VAR CONSTANT
	NULL:                                   			XWORD := 0;
	data:						iol_slave_bis00lh_data;			(*$	Parameters struct variable	$*)
	CONVERSION_this:			iol_slave;						(*$ Instance to which the method applies $*)
	
END_VAR



(*** Start parameter configuration ***)

(* STANDARD PARAMETERS CONFIGURATION *)

(* RMH RFID TEST *)
rfid_input_bitheader_1.CP := rfid_input_buffer.ByteArr[0].0;
rfid_input_bitheader_1.AA := rfid_input_buffer.ByteArr[0].1;
rfid_input_bitheader_1.AE := rfid_input_buffer.ByteArr[0].2;
rfid_input_bitheader_1.AF := rfid_input_buffer.ByteArr[0].3;
rfid_input_bitheader_1.Bit4 := rfid_input_buffer.ByteArr[0].4;
rfid_input_bitheader_1._TO := rfid_input_buffer.ByteArr[0].5;
rfid_input_bitheader_1.HF := rfid_input_buffer.ByteArr[0].6;
rfid_input_bitheader_1.BB := rfid_input_buffer.ByteArr[0].7;

rfid_input_bitheader_2.CP := rfid_input_buffer.ByteArr[0].0;
rfid_input_bitheader_2.AA := rfid_input_buffer.ByteArr[0].1;
rfid_input_bitheader_2.AE := rfid_input_buffer.ByteArr[0].2;
rfid_input_bitheader_2.AF := rfid_input_buffer.ByteArr[0].3;
rfid_input_bitheader_2.Bit4 := rfid_input_buffer.ByteArr[0].4;
rfid_input_bitheader_2._TO := rfid_input_buffer.ByteArr[0].5;
rfid_input_bitheader_2.HF := rfid_input_buffer.ByteArr[0].6;
rfid_input_bitheader_2.BB := rfid_input_buffer.ByteArr[0].7;

rfid_output_bitheader_1.TI := rfid_output_buffer.ByteArr[0].0;
rfid_output_bitheader_1.Bit1 := rfid_output_buffer.ByteArr[0].1;
rfid_output_bitheader_1.GR := rfid_output_buffer.ByteArr[0].2;
rfid_output_bitheader_1.Bit3 := rfid_output_buffer.ByteArr[0].3;
rfid_output_bitheader_1.Bit4 := rfid_output_buffer.ByteArr[0].4;
rfid_output_bitheader_1.KA := rfid_output_buffer.ByteArr[0].5;
rfid_output_bitheader_1.TI := rfid_output_buffer.ByteArr[0].6;
rfid_output_bitheader_1.Bit7 := rfid_output_buffer.ByteArr[0].7;

rfid_output_bitheader_2.TI := rfid_output_buffer.ByteArr[0].0;
rfid_output_bitheader_2.Bit1 := rfid_output_buffer.ByteArr[0].1;
rfid_output_bitheader_2.GR := rfid_output_buffer.ByteArr[0].2;
rfid_output_bitheader_2.Bit3 := rfid_output_buffer.ByteArr[0].3;
rfid_output_bitheader_2.Bit4 := rfid_output_buffer.ByteArr[0].4;
rfid_output_bitheader_2.KA := rfid_output_buffer.ByteArr[0].5;
rfid_output_bitheader_2.TI := rfid_output_buffer.ByteArr[0].6;
rfid_output_bitheader_2.Bit7 := rfid_output_buffer.ByteArr[0].7;


(*IF iol_slave_is_not_initialized(CONVERSION_this := CONVERSION_this)
	OR
	iol_slave_is_configured(CONVERSION_this := CONVERSION_this)
THEN
	RETURN;
END_IF


iol_slave_configure_parameter(
	current_value_address := ADR(CONVERSION_this.vendor_name),
	configured_value_address := NULL,
	length := SIZEOF(CONVERSION_this.vendor_name),
	_type := ADST_STRING,
	coe_index := 16#0010,
	coe_sub_index := 16#00,
	readable := TRUE,
	writeable := FALSE,
	to_check := FALSE,
	CONVERSION_this := CONVERSION_this);


iol_slave_configure_parameter(
	current_value_address := ADR(CONVERSION_this.product_name),
	configured_value_address := NULL,
	length := SIZEOF(CONVERSION_this.product_name),
	_type := ADST_STRING,
	coe_index := 16#0012,
	coe_sub_index := 16#00,
	readable := TRUE,
	writeable := FALSE,
	to_check := FALSE,
	CONVERSION_this := CONVERSION_this);

iol_slave_configure_parameter(
	current_value_address := ADR(CONVERSION_this.product_id),
	configured_value_address := NULL,
	length := SIZEOF(CONVERSION_this.product_id),
	_type := ADST_STRING,
	coe_index := 16#0013,
	coe_sub_index := 16#00,
	readable := TRUE,
	writeable := FALSE,
	to_check := FALSE,
	CONVERSION_this := CONVERSION_this);


iol_slave_configure_parameter(
	current_value_address := ADR(CONVERSION_this.hardware_revision),
	configured_value_address := NULL,
	length := SIZEOF(CONVERSION_this.hardware_revision),
	_type := ADST_STRING,
	coe_index := 16#0016,
	coe_sub_index := 16#00,
	readable := TRUE,
	writeable := FALSE,
	to_check := FALSE,
	CONVERSION_this := CONVERSION_this);

iol_slave_configure_parameter(
	current_value_address := ADR(CONVERSION_this.firmware_revision),
	configured_value_address := NULL,
	length := SIZEOF(CONVERSION_this.firmware_revision),
	_type := ADST_STRING,
	coe_index := 16#0017,
	coe_sub_index := 16#00,
	readable := TRUE,
	writeable := FALSE,
	to_check := FALSE,
	CONVERSION_this := CONVERSION_this);

iol_slave_configure_parameter(
	current_value_address := ADR(CONVERSION_this.current_app_specific_tag),
	configured_value_address := ADR(CONVERSION_this.configured_app_specific_tag),
	length := SIZEOF(CONVERSION_this.current_app_specific_tag),
	_type := ADST_STRING,
	coe_index := 16#0018,
	coe_sub_index := 16#00,
	readable := TRUE,
	writeable := TRUE,
	to_check := TRUE,
	CONVERSION_this := CONVERSION_this);
	
	

(* CUSTOM PARAMETERS CONFIGURATION *)
(*
iol_slave_configure_parameter(
	current_value_address := ADR(data.v_param_1),
	configured_value_address := ADR(data.v_param_1),
	length := SIZEOF(data.v_param_1),
	_type := ADST_UINT8,
	coe_index := 16#0040,
	coe_sub_index := 16#01,
	readable := TRUE,
	writeable := TRUE,
	to_check := FALSE,
	CONVERSION_this := CONVERSION_this);
	
iol_slave_configure_parameter(
	current_value_address := ADR(data.v_param_2),
	configured_value_address := ADR(data.v_param_2),
	length := SIZEOF(data.v_param_2),
	_type := ADST_UINT8,
	coe_index := 16#0040,
	coe_sub_index := 16#02,
	readable := TRUE,
	writeable := TRUE,
	to_check := FALSE,
	CONVERSION_this := CONVERSION_this);
	
iol_slave_configure_parameter(
	current_value_address := ADR(data.v_param_3),
	configured_value_address := ADR(data.v_param_3),
	length := SIZEOF(data.v_param_3),
	_type := ADST_UINT8,
	coe_index := 16#0040,
	coe_sub_index := 16#03,
	readable := TRUE,
	writeable := TRUE,
	to_check := FALSE,
	CONVERSION_this := CONVERSION_this);
	
iol_slave_configure_parameter(
	current_value_address := ADR(data.v_param_4),
	configured_value_address := ADR(data.v_param_4),
	length := SIZEOF(data.v_param_4),
	_type := ADST_UINT8,
	coe_index := 16#0040,
	coe_sub_index := 16#04,
	readable := TRUE,
	writeable := TRUE,
	to_check := FALSE,
	CONVERSION_this := CONVERSION_this);
	
iol_slave_configure_parameter(
	current_value_address := ADR(data.v_param_5),
	configured_value_address := ADR(data.v_param_5),
	length := SIZEOF(data.v_param_5),
	_type := ADST_UINT8,
	coe_index := 16#0040,
	coe_sub_index := 16#05,
	readable := TRUE,
	writeable := TRUE,
	to_check := FALSE,
	CONVERSION_this := CONVERSION_this);
	
iol_slave_configure_parameter(
	current_value_address := ADR(data.v_param_6),
	configured_value_address := ADR(data.v_param_6),
	length := SIZEOF(data.v_param_6),
	_type := ADST_UINT8,
	coe_index := 16#0040,
	coe_sub_index := 16#06,
	readable := TRUE,
	writeable := TRUE,
	to_check := FALSE,
	CONVERSION_this := CONVERSION_this);
	*)
	

	
CONVERSION_this.CONVERSION_private.last_info_data_index := 6;

(*** End parameter configuration ***)
iol_slave_configuration_completed(
	parameters_ptr := ADR(data),
	parameters_struct_size := SIZEOF(data),
	CONVERSION_this := CONVERSION_this);*)

END_FUNCTION

// ---- POUs/AFL extensions/IO_Link/FUN/iol_slave_ray26p_configure.TcPOU
(*$
<p>This function configures a generic <a target="_blank" href="#iol_slave">iol_slave</a> as a <strong>Sick WTB2SC - 2P3244</strong>. It allow to connect the object to the device-specific
parameters structure variable <a target="_blank" href="#iol_slave_wtb2sc_data">iol_slave_wtb2sc_data</a>.</p>
<p>This function should be called at startup only.</p>
$*)

FUNCTION iol_slave_ray26p_configure : VOID
VAR_IN_OUT
	data:					iol_slave_ray26p_data;			(*$	Parameters struct variable$*)
	CONVERSION_this:		iol_slave;						(*$ Instance to which the method applies $*)
END_VAR

VAR CONSTANT
	NULL:                                   			XWORD := 0;
END_VAR

IF iol_slave_is_not_initialized(CONVERSION_this := CONVERSION_this)
	OR
	iol_slave_is_configured(CONVERSION_this := CONVERSION_this)
THEN
	RETURN;
END_IF

(*** Start parameter configuration ***)

(* STANDARD PARAMETERS CONFIGURATION *)

iol_slave_configure_parameter(
	current_value_address := ADR(CONVERSION_this.vendor_name),
	configured_value_address := NULL,
	length := SIZEOF(CONVERSION_this.vendor_name),
	_type := ADST_STRING,
	coe_index := 16#0010,
	coe_sub_index := 16#00,
	readable := TRUE,
	writeable := FALSE,
	to_check := FALSE,
	CONVERSION_this := CONVERSION_this);

iol_slave_configure_parameter(
	current_value_address := ADR(CONVERSION_this.product_name),
	configured_value_address := NULL,
	length := SIZEOF(CONVERSION_this.product_name),
	_type := ADST_STRING,
	coe_index := 16#0012,
	coe_sub_index := 16#00,
	readable := TRUE,
	writeable := FALSE,
	to_check := FALSE,
	CONVERSION_this := CONVERSION_this);

iol_slave_configure_parameter(
	current_value_address := ADR(CONVERSION_this.product_id),
	configured_value_address := NULL,
	length := SIZEOF(CONVERSION_this.product_id),
	_type := ADST_STRING,
	coe_index := 16#0013,
	coe_sub_index := 16#00,
	readable := TRUE,
	writeable := FALSE,
	to_check := FALSE,
	CONVERSION_this := CONVERSION_this);


iol_slave_configure_parameter(
	current_value_address := ADR(CONVERSION_this.hardware_revision),
	configured_value_address := NULL,
	length := SIZEOF(CONVERSION_this.hardware_revision),
	_type := ADST_STRING,
	coe_index := 16#0016,
	coe_sub_index := 16#00,
	readable := TRUE,
	writeable := FALSE,
	to_check := FALSE,
	CONVERSION_this := CONVERSION_this);

iol_slave_configure_parameter(
	current_value_address := ADR(CONVERSION_this.firmware_revision),
	configured_value_address := NULL,
	length := SIZEOF(CONVERSION_this.firmware_revision),
	_type := ADST_STRING,
	coe_index := 16#0017,
	coe_sub_index := 16#00,
	readable := TRUE,
	writeable := FALSE,
	to_check := FALSE,
	CONVERSION_this := CONVERSION_this);


(* CUSTOM PARAMETERS CONFIGURATION *)

iol_slave_configure_parameter(
	current_value_address := ADR(data.teach_in_state),
	configured_value_address := NULL,
	length := SIZEOF(data.teach_in_state),
	_type := ADST_UINT8,
	coe_index := 16#003B,
	coe_sub_index :=16#00,
	readable := TRUE,
	writeable := FALSE,
	to_check := FALSE,
	CONVERSION_this := CONVERSION_this);
	
iol_slave_configure_parameter(
	current_value_address := ADR(data.teach_in_channel),
	configured_value_address := ADR(data.teach_in_channel),
	length := SIZEOF(data.teach_in_channel),
	_type := ADST_UINT8,
	coe_index := 16#003A,
	coe_sub_index :=16#00,
	readable := TRUE,
	writeable := TRUE,
	to_check := TRUE, (* to be evaluated *)
	CONVERSION_this := CONVERSION_this);
	
iol_slave_configure_parameter(
	current_value_address := ADR(data.sender_configuration),
	configured_value_address := ADR(data.sender_configuration),
	length := SIZEOF(data.sender_configuration),
	_type := ADST_UINT8,
	coe_index := 16#0061,
	coe_sub_index :=16#00,
	readable := TRUE,
	writeable := TRUE,
	to_check := TRUE, (* to be evaluated *)
	CONVERSION_this := CONVERSION_this);
	
iol_slave_configure_parameter(
	current_value_address := ADR(data.Pin2_configuration),
	configured_value_address := ADR(data.Pin2_configuration),
	length := SIZEOF(data.Pin2_configuration),
	_type := ADST_UINT8,
	coe_index := 16#0079,
	coe_sub_index :=16#00,
	readable := TRUE,
	writeable := TRUE,
	to_check := TRUE, (* to be evaluated *)
	CONVERSION_this := CONVERSION_this);

iol_slave_configure_parameter(
	current_value_address := ADR(data.quality_of_teach),
	configured_value_address := NULL,
	length := SIZEOF(data.quality_of_teach),
	_type := ADST_UINT8,
	coe_index := 16#0072,
	coe_sub_index :=16#00,
	readable := TRUE,
	writeable := FALSE,
	to_check := FALSE, (* to be evaluated *)
	CONVERSION_this := CONVERSION_this);
	
iol_slave_configure_parameter(
	current_value_address := ADR(data.system_state),
	configured_value_address := NULL,
	length := SIZEOF(data.system_state),
	_type := ADST_UINT8,
	coe_index := 16#00E2,
	coe_sub_index :=16#00,
	readable := TRUE,
	writeable := FALSE,
	to_check := FALSE, (* to be evaluated *)
	CONVERSION_this := CONVERSION_this);


CONVERSION_this.CONVERSION_private.last_info_data_index := 5;

(*** End parameter configuration ***)

iol_slave_configuration_completed(
	parameters_ptr := ADR(data),
	parameters_struct_size := SIZEOF(data),
	CONVERSION_this := CONVERSION_this);

END_FUNCTION

// ---- Application/CSP/Customer Interface/csp_customerInterfaces_old.TcPOU
 (*********************************** G.D S.p.A. - Technical Department ***********************************
============= PROGRAM INFO ============
FOLDER:             TBD
MACHINES INVOLVED:  TBD 

============= DESCRIPTION =============
Exit unit device declaration

============= REVISIONS ===============
Date		Version	 	Author      	Description             
----------	-------		------------  	--------------------------------------------
2019/03/27 	0000.00	 	CEC 			Creation of the PRG

**********************************************************************************************************)
(*$R process_ref:= prc; $*)

PROGRAM csp_customerInterfaces_old

VAR
	prc:								process;
	prc_path:							STRING;
	
	CasePacker:							csp_customerInterfaces_casePacker;
	Palletizer:							csp_customerInterfaces_palletizer;
	
END_VAR

VAR PERSISTENT
	Order:								csp_customerInterfaces_order;
	Product:							csp_customerInterfaces_product;
	Recipe:								csp_customerInterfaces_recipe;														
	Material:							ARRAY [0..14] OF csp_customerInterfaces_material;
	Mark:								csp_customerInterfaces_mark;
	NextOrder:							csp_customerInterfaces_order;	
	NextProduct:						csp_customerInterfaces_product;	
	NextRecipe:							csp_customerInterfaces_recipe;		
	NextMaterial:						ARRAY [0..14] OF csp_customerInterfaces_material;			
	MES:								csp_customerInterfaces_MES;	
		
END_VAR

_read_var_input();

_objects_manager();

IF NOT objects_running()
THEN
	RETURN;	
END_IF

_read_process_image();

_mode_manager();

CASE process_get_mode(prc) of
	MODE_ABSENT,
	MODE_INACTIVE:
		RETURN;
	MODE_TEST:
		_handle_process_test();
END_CASE

_set_runtime_properties();

(********************************* BODY *********************************)


(* CSP STATUS *)

Dock();
//CasePacker.Status.Online := machine_is_operational(csp.mch); 
//CasePacker.Status.Job := csp_main_brand.p_carton_format;
//CasePacker.Status.NextJob := // need to figure out next job
CasePacker.Status.Running := machine_is_running(csp.mch);

CasePacker.Status.Faulted.Main := machine_is_stopped(csp.mch)
									AND csp_main_interface.alarm_id_from_python <> 363 // CYCLE STOP FOR CASE SIDE
									AND csp_main_interface.alarm_id_from_python <> 622 // CYCLE STOP FOR TRANSFER SIDE
									AND csp_main_interface.alarm_id <> 363 // CYCLE STOP FOR CASE SIDE
									AND csp_main_interface.alarm_id <> 622; // CYCLE STOP FOR TRANSFER SIDE
									
CasePacker.Status.Faulted.CaseBlanks := csp_case_feed_magazine.AML_Faulted;

//CasePacker.Status.RunOut := csp_main_motorization.empty_command;
//CasePacker.Status.RunOutComplete := message_is_on(csp_case_virtualMaster.runout_complete);

CasePacker.Status.Rate.Target := LREAL_TO_INT(csp_main_motorization_manager.motm.actual_velocity_setpoint);
CasePacker.Status.Rate.Actual := LREAL_TO_INT(csp_main_motorization_manager.motm.actual_velocity);

CasePacker.Status.Stop.AutoReason := csp_main_interface.alarm_id; 
CasePacker.Status.Stop.Estop := machine_is_stop_emergency_active(csp.mch);
CasePacker.Status.Stop.Guard := NOT safety_integrated_series_is_safely_closed(csp_case_main_safety_guards.sis) OR NOT safety_integrated_series_is_safely_closed(csp_transfer_main_safety_guards.sis);
CasePacker.Status.Stop.Operator := message_is_on(csp_case_main_services_pushbuttons.stop_dchk.alarm_asm.message);

CasePacker.Status.Starved.CaseBlanks := message_is_on(csp_case_feed_magazine_level_zonemin.magazine_level_zone_min_wem);
CasePacker.Status.Starved.Glue := NOT digital_input_is_active(csp_case_glue_hotmelt.level_ok_di);
//CasePacker.Status.Starved.Labels :=
CasePacker.Status.Starved.Units := csp_transfer_infeed_clamp.min_prime;

CasePacker.Status.Blocked.Downstream := message_is_on(csp_case_discharge_reject_sensors.downstream_backup_hold_aem);
CasePacker.Status.Blocked.Reject := message_is_on(csp_case_discharge_reject_sensors.consecutive_blocked_reject_aem);
CasePacker.Status.Blocked.Waste := message_is_on(csp_transfer_crosspusher_reject.backup_di_dchk.alarm_asm.message);




 
(*
CasePacker.Start.PeakWait :=
CasePacker.Start.Ramp:=
CasePacker.Start.Request:=
CasePacker.Production.GoodCasesNoReset:=
CasePacker.Production.GoodPods:=
CasePacker.Production.GoodPodsNoReset:=*)
CasePacker.Production.GoodUnits:= csp_case_main_statistics.logsect.hmi_shift_independent_sampled_counters.total_good_products; //log_section_get_total_good_production(csp_case_main_statistics.logsect);
(*CasePacker.Production.GoodUnitsNoReset:=
CasePacker.Production.PercentScrapUnits:=
CasePacker.Production.Rejects.Infeed_waterfall:=
CasePacker.Production.Rejects.Accumulator:=
CasePacker.Production.Rejects.Case_Feed:=*)
CasePacker.Production.Rejects.Discharge:= csp_case_discharge_reject.Discharge_reject_count;
(*CasePacker.Production.Rejects.TBD5:=
CasePacker.Production.Rejects.TBD6:= *)
CasePacker.Production.TotalScrapUnits:= csp_case_main_statistics.logsect.hmi_shift_independent_sampled_counters.total_rejected; //log_section_get_total_rejected(csp_case_main_statistics.logsect);
CasePacker.Production.TotalUnits:= (CasePacker.Production.GoodUnits + CasePacker.Production.TotalScrapUnits);
(*CasePacker.Production.TotalUnitsNoReset:=

CasePacker.CaseBlanks.ConsumedCart:=
CasePacker.CaseBlanks.ConsumedTotal:=
CasePacker.Labels.Consumed:=
CasePacker.CtCall.FaultedCaseSupply:=csp_case_feed_magazine.AML_Faulted;
CasePacker.CtCall.FaultedMain:=machine_is_stopped(csp.mch);
CasePacker.CtCall.FullScrapBin:=
CasePacker.CtCall.LowCaseSupply:=csp_case_feed_magazine.Magazine_low_level;
CasePacker.CtCall.LowGlueSupply:=csp_case_glue_hotmelt.level_ok_di;
//CasePacker.CtCall.LowLabelSupply:=.
CasePacker.CtCall.TBD1:=
CasePacker.CtCall.TBD2:=
CasePacker.CtCall.TBD3:=
CasePacker.Dock[1].Active:=
CasePacker.Dock[1].AmrExited:=
CasePacker.Dock[1].DropAvailable:=
CasePacker.Dock[1].EntryAck:=
CasePacker.Dock[1].EntryOK:=
CasePacker.Dock[1].EntryReq:=
CasePacker.Dock[1].PickAvailable:=
*)

(************************************************************************)

_handle_messages();

_write_output();

ACTION _handle_messages:
;
END_ACTION

ACTION _handle_process_test:
;
END_ACTION

ACTION _mode_manager:
IF process_mode_req_is_pending(prc)
THEN
    process_apply_mode_req_first_step(prc);
    CASE process_get_mode(prc) OF
        MODE_TO_ABSENT:
			;
        MODE_TO_INACTIVE:
			;
        MODE_TO_TEST:
			;
        MODE_TO_OPERATIONAL:
			;
    END_CASE
    process_apply_mode_req_second_step(prc);
END_IF
END_ACTION

ACTION _objects_manager:
IF objects_initialization()
THEN
	process_init(
		object_name					:= 'csp_customerInterfaces.prc', 
		machine						:= csp.mch, 
		CONVERSION_this				:= prc);
		
	prc_path 						:= process_get_path(prc);
END_IF

IF objects_running()
THEN
	process_cycle(prc);
END_IF
END_ACTION

ACTION _read_process_image:
;
END_ACTION

ACTION _read_var_input:
;
END_ACTION

ACTION _set_runtime_properties:
//CasePacker.Status.Online := TRUE;
END_ACTION

ACTION _write_output:
;
END_ACTION

ACTION Dock:
//Flexlink to AMR Dock 1
CasePacker.Dock[1].DropAvailable:= csp_case_feed_magazine.Flexlink_to_AMR_DropAvailable_1;
CasePacker.Dock[1].PickAvailable:= csp_case_feed_magazine.Flexlink_to_AMR_PickAvailable_1; 
CasePacker.Dock[1].Active:= csp_case_feed_magazine.Flexlink_to_AMR_Active_1;
CasePacker.Dock[1].EntryAck:= csp_case_feed_magazine.Flexlink_to_AMR_EntryAck_1;
CasePacker.Dock[1].EntryOK:= csp_case_feed_magazine.Flexlink_to_AMR_EntryOK_1;

(*csp_case_feed_magazine.AMR_to_Flexlink_EntryReq_1*) RAJ_to_Flexlink[3].0:= CasePacker.Dock[1].EntryReq;
(*csp_case_feed_magazine.AMR_to_Flexlink_AmrExited_1*) RAJ_to_Flexlink[3].1:= CasePacker.Dock[1].AmrExited;

//Flexlink to AMR Dock 2
CasePacker.Dock[2].DropAvailable:= csp_case_feed_magazine.Flexlink_to_AMR_DropAvailable_2;
CasePacker.Dock[2].PickAvailable:= csp_case_feed_magazine.Flexlink_to_AMR_PickAvailable_2; 
CasePacker.Dock[2].Active:= csp_case_feed_magazine.Flexlink_to_AMR_Active_2;
CasePacker.Dock[2].EntryAck:= csp_case_feed_magazine.Flexlink_to_AMR_EntryAck_2;
CasePacker.Dock[2].EntryOK:= csp_case_feed_magazine.Flexlink_to_AMR_EntryOK_2;

(*csp_case_feed_magazine.AMR_to_Flexlink_EntryReq_2*) RAJ_to_Flexlink[3].2:= CasePacker.Dock[2].EntryReq;
(*csp_case_feed_magazine.AMR_to_Flexlink_AmrExited_2*) RAJ_to_Flexlink[3].3:= CasePacker.Dock[2].AmrExited;

//Flexlink to AMR Dock 3
CasePacker.Dock[3].DropAvailable:= csp_case_feed_magazine.Flexlink_to_AMR_DropAvailable_3;
CasePacker.Dock[3].PickAvailable:= csp_case_feed_magazine.Flexlink_to_AMR_PickAvailable_3; 
CasePacker.Dock[3].Active:= csp_case_feed_magazine.Flexlink_to_AMR_Active_3;
CasePacker.Dock[3].EntryAck:= csp_case_feed_magazine.Flexlink_to_AMR_EntryAck_3;
CasePacker.Dock[3].EntryOK:= csp_case_feed_magazine.Flexlink_to_AMR_EntryOK_3;

(*csp_case_feed_magazine.AMR_to_Flexlink_EntryReq_3*) RAJ_to_Flexlink[3].4:= CasePacker.Dock[3].EntryReq;
(*csp_case_feed_magazine.AMR_to_Flexlink_AmrExited_3*) RAJ_to_Flexlink[3].5:= CasePacker.Dock[3].AmrExited;
END_ACTION

END_PROGRAM

// ---- Application/CSP/Customer Interface/csp_customerInterfaces_old_2.TcPOU
 (*********************************** G.D S.p.A. - Technical Department ***********************************
============= PROGRAM INFO ============
FOLDER:             TBD
MACHINES INVOLVED:  TBD 

============= DESCRIPTION =============
Exit unit device declaration

============= REVISIONS ===============
Date		Version	 	Author      	Description             
----------	-------		------------  	--------------------------------------------
2019/03/27 	0000.00	 	CEC 			Creation of the PRG

**********************************************************************************************************)
(*$R process_ref:= prc; $*)

PROGRAM csp_customerInterfaces_old_2

VAR
	prc:								process;
	prc_path:							STRING;
	
	Order:								csp_customerInterfaces_order;
	Product:							csp_customerInterfaces_product;
	Recipe:								csp_customerInterfaces_recipe;														
	Material:							ARRAY [0..14] OF csp_customerInterfaces_material;
	Mark:								csp_customerInterfaces_mark;
	NextOrder:							csp_customerInterfaces_order;	
	NextProduct:						csp_customerInterfaces_product;	
	NextRecipe:							csp_customerInterfaces_recipe;		
	NextMaterial:						ARRAY [0..14] OF csp_customerInterfaces_material;			
	MES:								csp_customerInterfaces_MES;		
	CasePacker:							csp_customerInterfaces_casePacker;
	Palletizer:							csp_customerInterfaces_palletizer;
	

END_VAR

_read_var_input();

_objects_manager();

IF NOT objects_running()
THEN
	RETURN;	
END_IF

_read_process_image();

_mode_manager();

CASE process_get_mode(prc) of
	MODE_ABSENT,
	MODE_INACTIVE:
		RETURN;
	MODE_TEST:
		_handle_process_test();
END_CASE

_set_runtime_properties();

(********************************* BODY *********************************)


(* CSP STATUS *)

CasePacker.Status.Online := machine_is_operational(csp.mch); 
CasePacker.Status.Job := csp_main_brand.p_carton_format;
//CasePacker.Status.NextJob := // need to figure out next job
CasePacker.Status.Running := machine_is_running(csp.mch);

CasePacker.Status.Faulted.Main := machine_is_stopped(csp.mch)
									AND csp_main_interface.alarm_id_from_python <> 363 // CYCLE STOP FOR CASE SIDE
									AND csp_main_interface.alarm_id_from_python <> 622; // CYCLE STOP FOR TRANSFER SIDE
CasePacker.Status.Faulted.CaseBlanks := csp_case_feed_magazine.AML_Faulted;

CasePacker.Status.RunOut := csp_main_motorization.empty_command;
CasePacker.Status.RunOutComplete := message_is_on(csp_case_virtualMaster.runout_complete);

CasePacker.Status.Rate.Target := LREAL_TO_INT(csp_main_motorization_manager.motm.actual_velocity_setpoint);
CasePacker.Status.Rate.Actual := LREAL_TO_INT(csp_main_motorization_manager.motm.actual_velocity);

CasePacker.Status.Stop.AutoReason := csp_main_interface.alarm_id; 
CasePacker.Status.Stop.Estop := machine_is_stop_emergency_active(csp.mch);
CasePacker.Status.Stop.Guard := NOT safety_integrated_series_is_safely_closed(csp_case_main_safety_guards.sis) OR NOT safety_integrated_series_is_safely_closed(csp_transfer_main_safety_guards.sis);
CasePacker.Status.Stop.Operator := message_is_on(csp_case_main_services_pushbuttons.stop_dchk.alarm_asm.message);

CasePacker.Status.Starved.CaseBlanks := message_is_on(csp_case_feed_magazine_level_zonemin.magazine_level_zone_min_aem);
CasePacker.Status.Starved.Glue := NOT digital_input_is_active(csp_case_glue_hotmelt.level_ok_di);
//CasePacker.Status.Starved.Labels :=
CasePacker.Status.Starved.Units := csp_transfer_infeed_clamp.min_prime;

CasePacker.Status.Blocked.Downstream := message_is_on(csp_case_discharge_reject_sensors.downstream_backup_hold_aem);
CasePacker.Status.Blocked.Reject := message_is_on(csp_case_discharge_reject_sensors.consecutive_blocked_reject_aem);
CasePacker.Status.Blocked.Waste := message_is_on(csp_transfer_crosspusher_reject.backup_di_dchk.alarm_asm.message);

//Flexlink to AMR Dock 1
CasePacker.Dock[1].DropAvailable:= csp_case_feed_magazine.Flexlink_to_AMR_DropAvailable_1;
CasePacker.Dock[1].PickAvailable:= csp_case_feed_magazine.Flexlink_to_AMR_PickAvailable_1; 
CasePacker.Dock[1].Active:= csp_case_feed_magazine.Flexlink_to_AMR_Active_1;
CasePacker.Dock[1].EntryAck:= csp_case_feed_magazine.Flexlink_to_AMR_EntryAck_1;
CasePacker.Dock[1].EntryOK:= csp_case_feed_magazine.Flexlink_to_AMR_EntryOK_1;

(*csp_case_feed_magazine.AMR_to_Flexlink_EntryReq_1*) RAJ_to_Flexlink[3].0:= CasePacker.Dock[1].EntryReq;
(*csp_case_feed_magazine.AMR_to_Flexlink_AmrExited_1*) RAJ_to_Flexlink[3].1:= CasePacker.Dock[1].AmrExited;

//Flexlink to AMR Dock 2
CasePacker.Dock[2].DropAvailable:= csp_case_feed_magazine.Flexlink_to_AMR_DropAvailable_2;
CasePacker.Dock[2].PickAvailable:= csp_case_feed_magazine.Flexlink_to_AMR_PickAvailable_2; 
CasePacker.Dock[2].Active:= csp_case_feed_magazine.Flexlink_to_AMR_Active_2;
CasePacker.Dock[2].EntryAck:= csp_case_feed_magazine.Flexlink_to_AMR_EntryAck_2;
CasePacker.Dock[2].EntryOK:= csp_case_feed_magazine.Flexlink_to_AMR_EntryOK_2;

(*csp_case_feed_magazine.AMR_to_Flexlink_EntryReq_2*) RAJ_to_Flexlink[3].2:= CasePacker.Dock[2].EntryReq;
(*csp_case_feed_magazine.AMR_to_Flexlink_AmrExited_2*) RAJ_to_Flexlink[3].3:= CasePacker.Dock[2].AmrExited;

//Flexlink to AMR Dock 3
CasePacker.Dock[3].DropAvailable:= csp_case_feed_magazine.Flexlink_to_AMR_DropAvailable_3;
CasePacker.Dock[3].PickAvailable:= csp_case_feed_magazine.Flexlink_to_AMR_PickAvailable_3; 
CasePacker.Dock[3].Active:= csp_case_feed_magazine.Flexlink_to_AMR_Active_3;
CasePacker.Dock[3].EntryAck:= csp_case_feed_magazine.Flexlink_to_AMR_EntryAck_3;
CasePacker.Dock[3].EntryOK:= csp_case_feed_magazine.Flexlink_to_AMR_EntryOK_3;

(*csp_case_feed_magazine.AMR_to_Flexlink_EntryReq_3*) RAJ_to_Flexlink[3].4:= CasePacker.Dock[3].EntryReq;
(*csp_case_feed_magazine.AMR_to_Flexlink_AmrExited_3*) RAJ_to_Flexlink[3].5:= CasePacker.Dock[3].AmrExited;




 
(*

CasePacker.Start.PeakWait :=
CasePacker.Start.Ramp:=
CasePacker.Start.Request:=

CasePacker.Production.GoodCasesNoReset:=
CasePacker.Production.GoodPods:=
CasePacker.Production.GoodPodsNoReset:=
CasePacker.Production.GoodUnits:=
CasePacker.Production.GoodUnitsNoReset:=
CasePacker.Production.PercentScrapUnits:=
CasePacker.Production.Rejects.TBD1:=
CasePacker.Production.Rejects.TBD2:=
CasePacker.Production.Rejects.TBD3:=
CasePacker.Production.Rejects.TBD4:=
CasePacker.Production.Rejects.TBD5:=
CasePacker.Production.Rejects.TBD6:=
CasePacker.Production.TotalScrapUnits:=
CasePacker.Production.TotalUnits:=
CasePacker.Production.TotalUnitsNoReset:=

CasePacker.CaseBlanks.ConsumedCart:=
CasePacker.CaseBlanks.ConsumedTotal:=

CasePacker.Labels.Consumed:=

CasePacker.CtCall.FaultedCaseSupply:=csp_case_feed_magazine.AML_Faulted;
CasePacker.CtCall.FaultedMain:=machine_is_stopped(csp.mch);
CasePacker.CtCall.FullScrapBin:=
CasePacker.CtCall.LowCaseSupply:=csp_case_feed_magazine.Magazine_low_level;
CasePacker.CtCall.LowGlueSupply:=csp_case_glue_hotmelt.level_ok_di;
//CasePacker.CtCall.LowLabelSupply:=.
CasePacker.CtCall.TBD1:=
CasePacker.CtCall.TBD2:=
CasePacker.CtCall.TBD3:=

CasePacker.Dock[1].Active:=
CasePacker.Dock[1].AmrExited:=
CasePacker.Dock[1].DropAvailable:=
CasePacker.Dock[1].EntryAck:=
CasePacker.Dock[1].EntryOK:=
CasePacker.Dock[1].EntryReq:=
CasePacker.Dock[1].PickAvailable:=

*)

(************************************************************************)

_handle_messages();

_write_output();

ACTION _handle_messages:
;
END_ACTION

ACTION _handle_process_test:
;
END_ACTION

ACTION _mode_manager:
IF process_mode_req_is_pending(prc)
THEN
    process_apply_mode_req_first_step(prc);
    CASE process_get_mode(prc) OF
        MODE_TO_ABSENT:
			;
        MODE_TO_INACTIVE:
			;
        MODE_TO_TEST:
			;
        MODE_TO_OPERATIONAL:
			;
    END_CASE
    process_apply_mode_req_second_step(prc);
END_IF
END_ACTION

ACTION _objects_manager:
IF objects_initialization()
THEN
	process_init(
		object_name					:= 'csp_customerInterfaces.prc', 
		machine						:= csp.mch, 
		CONVERSION_this				:= prc);
		
	prc_path 						:= process_get_path(prc);
END_IF

IF objects_running()
THEN
	process_cycle(prc);
END_IF
END_ACTION

ACTION _read_process_image:
;
END_ACTION

ACTION _read_var_input:
;
END_ACTION

ACTION _set_runtime_properties:
;
END_ACTION

ACTION _write_output:
;
END_ACTION

END_PROGRAM

// ---- Application/CSP/Main/AccU Change/FB_RecoverPosition.TcPOU
FUNCTION_BLOCK FB_RecoverPosition
VAR_INPUT
	/// recover position - recovery position will be calculated prior to this being set true
	bRecover: BOOL;
	/// ex: 360*0.00000095367431640625
	lrScaling: LREAL;
	/// Absolute Encoder Pulses; Link to Position Feed Back Value Of The Drive
	diEncoderValue: DINT;
	/// Link To Persistent Variable; Current Encoder Position
	udiRetainedEncoderPos: UDINT;
	/// Link To Persistent Variable; Current Axis Position
	lrRetainedAxisPos: LREAL;
END_VAR
VAR_IN_OUT
	axis_ref: AXIS_REF;
END_VAR
VAR_OUTPUT
	lrRecovevedAxisPos: LREAL;
	bPositionRecovered: BOOL;
END_VAR
VAR
	udiPwrUpEncoderPos: UDINT;
	lrMaxPosAtEncRollOver: LREAL;
	udiRollPosition: UDINT;
	lrRollCorrection: LREAL;
	lrPwrOffDistance: LREAL;
	/// Maximum Count of Absolute Encoder Pulses
	cudiMaxEncoderCount: UDINT := 4294967295;
	cudiHalfMaxCount: UDINT := 2147483647;
	mcSetPosition: MC_SetPosition;
END_VAR

udiPwrUpEncoderPos := DINT_TO_UDINT(diEncoderValue);
lrRollCorrection := 0;
lrMaxPosAtEncRollOver := UDINT_TO_LREAL(cudiMaxEncoderCount) * lrScaling;

// Find Roll Over/Under Position
IF udiRetainedEncoderPos > cudiHalfMaxCount THEN
	// Roll Over
	udiRollPosition := udiRetainedEncoderPos - cudiHalfMaxCount;
	IF udiPwrUpEncoderPos <= udiRollPosition THEN
		lrRollCorrection := lrMaxPosAtEncRollOver;
	END_IF
ELSE
	// Roll Under
	udiRollPosition := udiRetainedEncoderPos + cudiHalfMaxCount;
	IF udiPwrUpEncoderPos >= udiRollPosition THEN
		lrRollCorrection := -1.0 * lrMaxPosAtEncRollOver;
	END_IF		
END_IF

// How Far Did Encoder Move During Power Off
IF udiPwrUpEncoderPos > udiRetainedEncoderPos THEN
	lrPwrOffDistance := UDINT_TO_LREAL(udiPwrUpEncoderPos - udiRetainedEncoderPos) * lrScaling;
ELSE
	lrPwrOffDistance := -1.0 * UDINT_TO_LREAL(udiRetainedEncoderPos - udiPwrUpEncoderPos) * lrScaling;
END_IF

// Recovered Axis Position
lrRecovevedAxisPos := lrRetainedAxisPos + lrPwrOffDistance + lrRollCorrection;


mcSetPosition(
	Axis:= axis_ref, 
	Execute:= bRecover, 
	Position:= lrRecovevedAxisPos, 
	Mode:= FALSE, // absolute 
	Options:= , 
	Done=> bPositionRecovered, 
	Busy=> , 
	Error=> , 
	ErrorID=> );

END_FUNCTION_BLOCK

// ---- Application/CSP/Main/csp_main_old.TcPOU
(*********************************** G.D S.p.A. - Technical Department ***********************************
============= PROGRAM INFO ============
FOLDER:             TBD
MACHINES INVOLVED:  TBD 

============= DESCRIPTION =============
csp main program

============= REVISIONS ===============
Date		Version	 	Author      	Description             
----------	-------		------------  	--------------------------------------------
2019/04/05 	0000.00	 	M.Grasso		Creation of the PRG

**********************************************************************************************************)
(*$R
	process_ref := prc;
$*)
PROGRAM csp_main_old
VAR
	prc:												process;
	prc_path:											STRING;
		
	cabinet_ethercat_master:							net_ethercat_master;
	cabinet_transfer_ethercat_master:					net_ethercat_master;
	
	is_SFI:												BOOL := TRUE;
	
END_VAR

VAR_INPUT
	
	i_cabinet_is_running:								BOOL;
	
	i_machine_motor_axis_ref:							POINTER TO axis;
	
	i_csp_data_ref:										POINTER TO csp_customerInterfaces_casePacker;	
	i_start_job_request:								BOOL;	
	i_cycle_enable_request:								BOOL;
	i_end_job_request:									BOOL;	
	i_order_information:								POINTER TO csp_customerInterfaces_order;
	i_product_information:								POINTER TO csp_customerInterfaces_product;
	i_recipe_information:								POINTER TO csp_customerInterfaces_recipe;
	i_current_material_information:						POINTER TO ARRAY[0..14] OF csp_customerInterfaces_material;
	i_next_material_information:						POINTER TO ARRAY[0..14] OF csp_customerInterfaces_material;	
	i_mark_bubd_information:							POINTER TO csp_customerInterfaces_markBUBD;	
	i_cartons_count:									DINT;
	i_next_recipe_information:							POINTER TO csp_customerInterfaces_recipe;
	
	(*mch interface*)
	i_cartoner_RunOutComplete:							BOOL;
	i_filler_upstream_coffee:							BOOL;

END_VAR

VAR_OUTPUT
	o_reset_button:										BOOL;
	o_start_button:										BOOL;
END_VAR

_read_var_input();

_object_manager();

IF NOT objects_running()
THEN
	RETURN;	
END_IF

_read_process_image();

_mode_manager();

CASE process_get_mode(prc) of
	MODE_ABSENT,
	MODE_INACTIVE:
		RETURN;
	MODE_TEST:
		_handle_process_test();
END_CASE

_set_runtime_properties();

(********************************* BODY *********************************)

(************************************************************************)

_handle_messages();

_write_output();

ACTION _handle_messages:
;
END_ACTION

ACTION _handle_process_test:
;
END_ACTION

ACTION _mode_manager:
IF process_mode_req_is_pending(prc)
THEN
    process_apply_mode_req_first_step(prc);
    CASE process_get_mode(prc) OF
        MODE_TO_ABSENT:
			;
        MODE_TO_INACTIVE:
			;
        MODE_TO_TEST:
			;
        MODE_TO_OPERATIONAL:
			;
    END_CASE
    process_apply_mode_req_second_step(prc);
END_IF
END_ACTION

ACTION _object_manager:
IF net_initialization()
THEN
		
	net_ethercat_master_init(
		object_name 				:= CONCAT(prc_path, '_cabinet_ethercat_master'), 
		hw_connected				:= TRUE, 
		process						:= prc, 
		CONVERSION_this				:= cabinet_ethercat_master);
		
(*	net_ethercat_master_init(
		object_name 				:= CONCAT(prc_path, '_cabinet_case_ethercat_master'), 
		hw_connected				:= FALSE, 
		process						:= prc, 
		CONVERSION_this				:= cabinet_case_ethercat_master);*)

net_ethercat_master_init(
		object_name 				:= CONCAT(prc_path, '_cabinet_transfer_ethercat_master'), 
		hw_connected				:= TRUE, 
		process						:= prc, 
		CONVERSION_this				:= cabinet_transfer_ethercat_master);				

	
END_IF


IF objects_initialization()
THEN
	process_init(
		object_name					:= 'csp_main.prc', 
		machine						:= csp.mch, 
		CONVERSION_this				:= prc);
		
	prc_path 						:= process_get_path(prc);
	
	hmi_init(
		hmi_is_required				:= TRUE, 
		plc_hmi_protocol_enable		:= FALSE, 
		process						:= prc);
END_IF

IF objects_running()
THEN
	process_cycle(prc);
END_IF
END_ACTION

ACTION _read_process_image:
;
END_ACTION

ACTION _read_var_input:
i_machine_motor_axis_ref				:= 	ADR(csp_main_motorization_virtualManager.virtual_master_test); //TODO: this will need an update

i_csp_data_ref							:= 	ADR(csp_customerInterfaces.CasePacker);
i_start_job_request						:= 	csp_customerInterfaces.MES.StartJobReq;
i_cycle_enable_request					:= 	csp_customerInterfaces.MES.CycleEnable;
i_end_job_request						:= 	csp_customerInterfaces.MES.EndJobReq;
i_order_information						:= 	ADR(csp_customerInterfaces.Order);
i_product_information					:= 	ADR(csp_customerInterfaces.Product);
i_recipe_information					:= 	ADR(csp_customerInterfaces.Recipe);
i_current_material_information			:= 	ADR(csp_customerInterfaces.Material);
i_next_material_information				:= 	ADR(csp_customerInterfaces.NextMaterial);	
i_mark_bubd_information					:= 	ADR(csp_customerInterfaces.Mark.BUBD);
i_cartons_count							:=	csp_transfer_infeed_metering_jam.cartons_count;
i_next_recipe_information				:= ADR(csp_customerInterfaces.NextRecipe);
END_ACTION

ACTION _set_runtime_properties:
;
END_ACTION

ACTION _write_output:
o_reset_button	:= csp_case_main_services_pushbuttons.reset_pressed OR csp_transfer_main_services_pushbuttons.reset_pressed;
o_start_button	:= 
	(
		csp_case_main_services_pushbuttons.start_pressed
	 	OR
		csp_transfer_main_services_pushbuttons.start_pressed
	)
	AND
	not csp_main_jogManager.jog_is_active;
END_ACTION

END_PROGRAM

// ---- Application/CSP/Main/csp_main_old_2.TcPOU
(*********************************** G.D S.p.A. - Technical Department ***********************************
============= PROGRAM INFO ============
FOLDER:             TBD
MACHINES INVOLVED:  TBD 

============= DESCRIPTION =============
csp main program

============= REVISIONS ===============
Date		Version	 	Author      	Description             
----------	-------		------------  	--------------------------------------------
2019/04/05 	0000.00	 	M.Grasso		Creation of the PRG

**********************************************************************************************************)
(*$R
	process_ref := prc;
$*)
PROGRAM csp_main_old_2
VAR
	prc:												process;
	prc_path:											STRING;
		
	cabinet_ethercat_master:							net_ethercat_master;
	cabinet_transfer_ethercat_master:					net_ethercat_master;
	
	is_SFI:												BOOL := TRUE;
	
END_VAR

VAR_INPUT
	
	i_cabinet_is_running:								BOOL;
	
	i_machine_motor_axis_ref:							POINTER TO axis;

END_VAR

VAR_OUTPUT
	o_reset_button:										BOOL;
	o_start_button:										BOOL;
END_VAR

_read_var_input();

_object_manager();

IF NOT objects_running()
THEN
	RETURN;	
END_IF

_read_process_image();

_mode_manager();

CASE process_get_mode(prc) of
	MODE_ABSENT,
	MODE_INACTIVE:
		RETURN;
	MODE_TEST:
		_handle_process_test();
END_CASE

_set_runtime_properties();

(********************************* BODY *********************************)

(************************************************************************)

_handle_messages();

_write_output();

ACTION _handle_messages:
;
END_ACTION

ACTION _handle_process_test:
;
END_ACTION

ACTION _mode_manager:
IF process_mode_req_is_pending(prc)
THEN
    process_apply_mode_req_first_step(prc);
    CASE process_get_mode(prc) OF
        MODE_TO_ABSENT:
			;
        MODE_TO_INACTIVE:
			;
        MODE_TO_TEST:
			;
        MODE_TO_OPERATIONAL:
			;
    END_CASE
    process_apply_mode_req_second_step(prc);
END_IF
END_ACTION

ACTION _object_manager:
IF net_initialization()
THEN
		
	net_ethercat_master_init(
		object_name 				:= CONCAT(prc_path, '_cabinet_ethercat_master'), 
		hw_connected				:= TRUE, 
		process						:= prc, 
		CONVERSION_this				:= cabinet_ethercat_master);
		
(*	net_ethercat_master_init(
		object_name 				:= CONCAT(prc_path, '_cabinet_case_ethercat_master'), 
		hw_connected				:= FALSE, 
		process						:= prc, 
		CONVERSION_this				:= cabinet_case_ethercat_master);*)

net_ethercat_master_init(
		object_name 				:= CONCAT(prc_path, '_cabinet_transfer_ethercat_master'), 
		hw_connected				:= TRUE, 
		process						:= prc, 
		CONVERSION_this				:= cabinet_transfer_ethercat_master);				

	
END_IF


IF objects_initialization()
THEN
	process_init(
		object_name					:= 'csp_main.prc', 
		machine						:= csp.mch, 
		CONVERSION_this				:= prc);
		
	prc_path 						:= process_get_path(prc);
	
	hmi_init(
		hmi_is_required				:= TRUE, 
		plc_hmi_protocol_enable		:= FALSE, 
		process						:= prc);
END_IF

IF objects_running()
THEN
	process_cycle(prc);
END_IF
END_ACTION

ACTION _read_process_image:
;
END_ACTION

ACTION _read_var_input:
//i_cabinet_is_running					:= cb.o_machine_is_running; (*MARCO*)
i_machine_motor_axis_ref				:= ADR(csp_main_motorization_virtualManager.virtual_master_test); //TODO: this will need an update
END_ACTION

ACTION _set_runtime_properties:
;
END_ACTION

ACTION _write_output:
o_reset_button	:= csp_case_main_services_pushbuttons.reset_pressed OR csp_transfer_main_services_pushbuttons.reset_pressed;
o_start_button	:= 
	(
		csp_case_main_services_pushbuttons.start_pressed
	 	OR
		csp_transfer_main_services_pushbuttons.start_pressed
	)
	AND
	not csp_main_jogManager.jog_is_active;
END_ACTION

END_PROGRAM

// ---- Application/CSP/Main/Phase Manager/csp_main_phaseManager_near_end_run.TcPOU
(*********************************** G.D S.p.A. - Technical Department ***********************************
============= PROGRAM INFO ============
FOLDER:             TBD
MACHINES INVOLVED:  TBD 

============= DESCRIPTION =============
WN phase manager program

============= REVISIONS ===============
Date		Version	 	Author      	Description             
----------	-------		------------  	--------------------------------------------
2021/03/18 	0000.01	 	S.Uccellari 	Creation of the PRG
**********************************************************************************************************)
(*$R
	process_ref := prc;
$*)
PROGRAM csp_main_phaseManager_near_end_run
VAR
	prc:												process;
	prc_path:											STRING;
	
	fsm_enable_conditions:								BOOL;
	fsm_status:											INT;
	
	near_end_run_running:								BOOL;
	near_end_run_done:									BOOL;
	
	square_wave_dvr:									BOOL;
	square_wave_rtrig:									R_TRIG;
	cups_done_cnt:										DINT;	
	cups_to_be_done_npr:								DINT;	(*$P desc := near end of run - cups to be done; $*)
	hmi_cups_remaining_nvr:								DINT;	(*$M $*)
	
END_VAR

_read_var_input();

_object_manager();

IF NOT objects_running()
THEN
	RETURN;	
END_IF

_read_process_image();

_mode_manager();

CASE process_get_mode(prc) of
	MODE_ABSENT,
	MODE_INACTIVE:
		RETURN;
	MODE_TEST:
		_handle_process_test();
END_CASE

_set_runtime_properties();

(********************************* BODY *********************************)

(************************************************************************)

(**************************** PROGRAM HANDLER ***************************)
run_cycle();
(************************************************************************)

_handle_messages();

_write_output();

ACTION _handle_messages:
;
END_ACTION

ACTION _handle_process_test:
;
END_ACTION

ACTION _mode_manager:
IF process_mode_req_is_pending(prc)
THEN
    process_apply_mode_req_first_step(prc);
    CASE process_get_mode(prc) OF
        MODE_TO_ABSENT:
			;
        MODE_TO_INACTIVE:
			;
        MODE_TO_TEST:
			;
        MODE_TO_OPERATIONAL:
			;
    END_CASE
    process_apply_mode_req_second_step(prc);
END_IF
END_ACTION

ACTION _object_manager:
IF objects_initialization()
THEN
	sub_process_init(
		object_name					:= 'csp_main_phaseManager_near_end_run.prc', 
		process						:= csp_main_phaseManager.prc, 
		CONVERSION_this				:= prc);
		
	prc_path 						:= process_get_path(prc);


END_IF

IF objects_running()
THEN
	process_cycle(prc);
END_IF
END_ACTION

ACTION _read_process_image:
;
END_ACTION

ACTION _read_var_input:
;
END_ACTION

ACTION _set_runtime_properties:
;
END_ACTION

ACTION _write_output:
;
END_ACTION

ACTION run_cycle:
IF	csp_main_phaseManager.fsm_status = CSP_MAIN_PHASE_MANAGER_STATUS_UNDEFINED_0
	AND
	csp_main_phaseManager.p_mes_interface_enable
THEN	
	fsm_status := 0;
END_IF

fsm_enable_conditions :=
	(
		csp_main_phaseManager.fsm_status
		=
		CSP_MAIN_PHASE_MANAGER_STATUS_NEAR_END_OF_RUN_50
	);
	
IF	NOT fsm_enable_conditions
	AND
	near_end_run_running	
THEN
	fsm_status := 666;
END_IF

CASE fsm_status OF
	0:
		IF fsm_enable_conditions
		THEN
			near_end_run_done := FALSE;
			near_end_run_running := TRUE;
			cups_done_cnt := 0;		
			fsm_status := 10;
		END_IF
		
	10:
		//square_wave_dvr := axis_get_actual_modulo_position(csp_main_motorization_machineMotor.encoder_axis_720) > 360;
		square_wave_rtrig(CLK := square_wave_dvr);
		
		//MARCO 1204
		(*
		IF square_wave_rtrig.Q
		THEN
			IF	shift_register_step_has_status_item(
				step_id						:= csp_exitUnit_shiftRegister.SHIFT_LAST_STEP,
				status_bits_to_be_true		:= ITEM_HAS_COFFEE,
				status_bits_to_be_false		:= NONE,
				CONVERSION_this				:= csp_exitUnit_shiftRegister.lineA_sr)
			THEN				
				cups_done_cnt := cups_done_cnt + 1;					
			END_IF	
			IF	shift_register_step_has_status_item(
				step_id						:= csp_exitUnit_shiftRegister.SHIFT_LAST_STEP,
				status_bits_to_be_true		:= ITEM_HAS_COFFEE,
				status_bits_to_be_false		:= NONE,
				CONVERSION_this				:= csp_exitUnit_shiftRegister.lineB_sr)
			THEN				
				cups_done_cnt := cups_done_cnt + 1;					
			END_IF			
		END_IF

		IF  cups_done_cnt >= cups_to_be_done_npr
		THEN
			hmi_cups_remaining_nvr := 0;	
			fsm_status :=	555;	
		ELSE
			hmi_cups_remaining_nvr := cups_to_be_done_npr - cups_done_cnt;	
		END_IF
		
		csp_main.i_csp_data_ref^.Production.RemainingPods := hmi_cups_remaining_nvr;
		
		*)

	555:
		near_end_run_running := FALSE;
		near_end_run_done := TRUE;
		
		//IF	NOT csp_main.i_upstream_coffee^.SiloLow //MARCO 0904
		//THEN
			near_end_run_running := FALSE;
			near_end_run_done := FALSE;
			fsm_status := 0;
		//END_IF		
		
	666:
		near_end_run_running := FALSE;
		near_end_run_done := FALSE;
		
		//IF NOT csp_main.i_upstream_coffee^.SiloLow //MARCO 0904
		//THEN
			fsm_status := 0;
		//END_IF
END_CASE
END_ACTION

END_PROGRAM

// ---- Application/CSP/Main/Safety/Drives/csp_main_safety_drives_commonConfiguration.TcPOU
(*********************************** G.D S.p.A. - Technical Department ***********************************
============= PROGRAM INFO ============
FOLDER:             TBD
MACHINES INVOLVED:  TBD 

============= DESCRIPTION =============
Machine drives common configurations

============= REVISIONS ===============
Date		Version	 	Author      	Description             
----------	-------		------------  	--------------------------------------------
2019/07/24 	0000.00	 	M.Grasso		Creation of the PRG

**********************************************************************************************************)

PROGRAM csp_main_safety_drives_commonConfiguration
VAR
	prc:					process;
	prc_path:				STRING;
	
	sig:					safety_integrated_group;
	rack_smes_sis:			safety_integrated_series;
	standalone_smes_sis:	safety_integrated_series;
	smm1_sis:				safety_integrated_series;
END_VAR

_read_var_input();

_object_manager();

IF NOT objects_running()
THEN
	RETURN;	
END_IF

_read_process_image();

_mode_manager();

CASE process_get_mode(prc) OF
	MODE_ABSENT,
	MODE_INACTIVE:
		RETURN;
	MODE_TEST:
		_handle_process_test();
END_CASE

_set_runtime_properties();

(********************************* BODY *********************************)
IF descriptor_get_reset_edge(prc.descriptor)
THEN
	safety_integrated_series_close(rack_smes_sis);
	safety_integrated_series_close(standalone_smes_sis);
END_IF
(************************************************************************)

_handle_messages();

_write_output();

ACTION _handle_messages:
;
END_ACTION

ACTION _handle_process_test:
;
END_ACTION

ACTION _mode_manager:
IF process_mode_req_is_pending(prc)
THEN
    process_apply_mode_req_first_step(prc);
    CASE process_get_mode(prc) OF
        MODE_TO_ABSENT:
			;
        MODE_TO_INACTIVE:
			;
        MODE_TO_TEST:
			;
        MODE_TO_OPERATIONAL:
			;
    END_CASE
    process_apply_mode_req_second_step(prc);
END_IF
END_ACTION

ACTION _object_manager:
IF objects_initialization()
THEN
	sub_process_init(
		object_name					:= 'csp_main_safety_drives_commonConfiguration.prc', 
		process						:= csp_main_safety_drives.prc, 
		CONVERSION_this				:= prc);
		
	prc_path 						:= process_get_path(prc);
	
	(*
	(* SIG *)
	safety_integrated_group_init(
		object_name					:=	CONCAT(prc_path, '_sig'),
		controller					:=	sw_configurator.WU_INTERFACE.drives_safety_controller_ref^,
		process						:=	prc,
		CONVERSION_this				:=	sig);	
		
	(* DRIVES RACK SERIES *)
	safety_integrated_series_init(
		object_name					:=	CONCAT(prc_path, '_rack_smes_sis'),
		_type						:=	SAFETY_INTEGRATED_SERIES_TYPE_RESET,
		discrepancy_active			:=	FALSE,
		forced_open_active			:=	TRUE,
		process						:=	prc,
		conversion_this				:=	rack_smes_sis);

	safety_integrated_series_add_safety_integrated_group(
		group						:=	sig,
		CONVERSION_this				:=	rack_smes_sis);

	safety_integrated_series_add_safety_integrated_series(
		series_active				:=	TRUE,
		series_polarity_direct		:=	TRUE,
		contact						:=	wu_main_safety_drives_powerSupply.sis,
		CONVERSION_this				:=	rack_smes_sis);	

	(* STANDALONE DRIVES SERIES *)
	safety_integrated_series_init(
		object_name					:=	CONCAT(prc_path, '_standalone_smes__sis'),
		_type						:=	SAFETY_INTEGRATED_SERIES_TYPE_RESET,
		discrepancy_active			:=	FALSE,
		forced_open_active			:=	TRUE,
		process						:=	prc,
		conversion_this				:=	standalone_smes_sis);

	safety_integrated_series_add_safety_integrated_group(
		group						:=	sig,
		CONVERSION_this				:=	standalone_smes_sis);

	safety_integrated_series_add_safety_integrated_series(
		series_active				:=	TRUE,
		series_polarity_direct		:=	TRUE,
		contact						:=	sw_configurator.WU_INTERFACE.delayed_emergency_series_ref^,
		CONVERSION_this				:=	standalone_smes_sis);			
	
	(* COMMON SMM1 *)		
	safety_integrated_series_init(
		object_name					:=	CONCAT(prc_path, '_smm1_sis'),
		_type						:=	SAFETY_INTEGRATED_SERIES_TYPE_RESET,
		discrepancy_active			:=	FALSE,
		forced_open_active			:=	TRUE,
		process						:=	prc,
		CONVERSION_this				:=	smm1_sis);

	safety_integrated_series_add_safety_integrated_group(
		group						:=	sig,
		CONVERSION_this				:=	smm1_sis);

	safety_integrated_series_add_safety_integrated_series(
		series_active 				:= TRUE,
		series_polarity_direct 		:= TRUE,
		contact 					:= wu_main_safety_handwheel.sis,
        CONVERSION_this 			:= smm1_sis);	
*)	
END_IF

IF objects_running()
THEN
	process_cycle(prc);
	
	safety_integrated_group_cycle(sig);
	safety_integrated_series_cycle(rack_smes_sis);
	safety_integrated_series_cycle(standalone_smes_sis);
	safety_integrated_series_cycle(smm1_sis);
END_IF
END_ACTION

ACTION _read_process_image:
;
END_ACTION

ACTION _read_var_input:
;
END_ACTION

ACTION _set_runtime_properties:
;
END_ACTION

ACTION _write_output:
;
END_ACTION

END_PROGRAM

// ---- Application/CSP/Main/Safety/Drives/csp_main_safety_drives_powerSupply.TcPOU
(*********************************** G.D S.p.A. - Technical Department ***********************************
============= PROGRAM INFO ============
FOLDER:             TBD
MACHINES INVOLVED:  TBD 

============= DESCRIPTION =============

============= REVISIONS ===============
Date		Version	 	Author      	Description             
----------	-------		------------  	--------------------------------------------
2019/04/09 	0000.00	 	M.Grasso		Creation of the PRG

**********************************************************************************************************)
(*$R process_ref:= prc; $*)

PROGRAM csp_main_safety_drives_powerSupply
VAR
	prc:												process;
	prc_path:											STRING;
	
	sig:												safety_integrated_group;
	sis:												safety_integrated_series;	
END_VAR

_read_var_input();

_objects_manager();

IF NOT objects_running()
THEN
	RETURN;	
END_IF

_read_process_image();

_mode_manager();

CASE process_get_mode(prc) OF
	MODE_ABSENT,
	MODE_INACTIVE:
		RETURN;
	MODE_TEST:
		;
END_CASE

_set_runtime_properties();

(********************************* BODY *********************************)
safety_integrated_series_close(sis);
(************************************************************************)

_handle_messages();

_write_output();

ACTION _handle_messages:
;
END_ACTION

ACTION _handle_process_test:
;
END_ACTION

ACTION _mode_manager:
IF process_mode_req_is_pending(prc)
THEN
    process_apply_mode_req_first_step(prc);
    CASE process_get_mode(prc) OF
        MODE_TO_ABSENT:
			;
        MODE_TO_INACTIVE:
			;
        MODE_TO_TEST:
			;
        MODE_TO_OPERATIONAL:
			;
    END_CASE
    process_apply_mode_req_second_step(prc);
END_IF
END_ACTION

ACTION _objects_manager:
IF objects_initialization()
THEN

	sub_process_init(
		object_name				:= 'csp_main_safety_drives_powerSupply.prc', 
		process					:= csp_main_safety_drives.prc, 
		CONVERSION_this			:= prc);
		
	prc_path 					:= process_get_path(prc);
	
	

END_IF
IF	objects_running()
THEN
    process_cycle(prc);

END_IF
END_ACTION

ACTION _read_process_image:
;
END_ACTION

ACTION _read_var_input:
;
END_ACTION

ACTION _set_runtime_properties:
;
END_ACTION

ACTION _write_output:
;
END_ACTION

END_PROGRAM

// ---- Application/CSP/Main/Safety/Emergency/csp_main_safety_emergency.TcPOU
(*********************************** G.D S.p.A. - Technical Department ***********************************
============= PROGRAM INFO ============
FOLDER:             TBD
MACHINES INVOLVED:  TBD 

============= DESCRIPTION =============
Machine notaus series

============= REVISIONS ===============
Date		Version	 	Author      	Description             
----------	-------		------------  	--------------------------------------------
2020/02/10 	0000.00	 	M.Grasso		Creation of the PRG

**********************************************************************************************************)
(*$R process_ref:= prc; $*)

PROGRAM csp_main_safety_emergency
VAR
	prc:											process;
	prc_path:										STRING;
	
 END_VAR

_read_var_input();

_objects_manager();

IF NOT objects_running()
THEN
	RETURN;	
END_IF

_read_process_image();

_mode_manager();

CASE process_get_mode(prc) OF
	MODE_ABSENT,
	MODE_INACTIVE:
		RETURN;
	MODE_TEST:
		;
END_CASE

_set_runtime_properties();

(********************************* BODY *********************************)
IF	descriptor_get_reset_edge(prc.descriptor)
THEN
	safety_integrated_series_close(sis);
	safety_integrated_series_close(delayed_sis);
END_IF
(************************************************************************)

_handle_messages();

_write_output();

ACTION _handle_messages:
;
END_ACTION

ACTION _handle_process_test:
;
END_ACTION

ACTION _mode_manager:
IF process_mode_req_is_pending(prc)
THEN
    process_apply_mode_req_first_step(prc);
    CASE process_get_mode(prc) OF
        MODE_TO_ABSENT:
			;
        MODE_TO_INACTIVE:
			;
        MODE_TO_TEST:
			;
        MODE_TO_OPERATIONAL:
			;
    END_CASE
    process_apply_mode_req_second_step(prc);
END_IF
END_ACTION

ACTION _objects_manager:
IF objects_initialization()
THEN

	sub_process_init(
		object_name								:= 'csp_main_safety_emergency.prc', 
		process									:= csp_main_safety.prc, 
		CONVERSION_this							:= prc);
		
	prc_path 									:= process_get_path(prc);

END_IF


IF	objects_running()
THEN
    process_cycle(prc);
END_IF
END_ACTION

ACTION _read_process_image:
;
END_ACTION

ACTION _read_var_input:
;
END_ACTION

ACTION _set_runtime_properties:
;
END_ACTION

ACTION _write_output:
;
END_ACTION

END_PROGRAM

// ---- Application/CSP/Main/Services/RFID FB/FB_BIS00LH.TcPOU
FUNCTION_BLOCK FB_BIS00LH
VAR_IN_OUT
	IO: ST_BIS00LH_IO;
END_VAR
VAR_INPUT
	///	iDevice : ST_Alarm2;
	ReadMode: BOOL;
	WriteCMode: BOOL;
	GroundStateRequest: BOOL;
	ShutdownRequest: BOOL;
	StartAddress: UINT;
	NumberOfBytes: UINT;
	WC_Value: BYTE;
	NumTags: INT;
	RecipeValue: BYTE;
END_VAR
VAR_IN_OUT
	/// 0-255 range
	//Cam: ST_Cam;
END_VAR
VAR_OUTPUT
	DeviceReadyBB: BOOL;
	TagPresentCP: BOOL;
	JobAcceptedAA: BOOL;
	JobEndAE: BOOL;
	JobErrorAF: BOOL;
	ToggleTO: BOOL;
	HeadFailureHF: BOOL;
	JobOk: BOOL;
	WriteOK: BOOL;
	ReadOK: BOOL;
	Error: BOOL;
	ER: BOOL;
	CP: BOOL;
	AA: BOOL;
	AF: BOOL;
	BB: BOOL;
	ValueRead: BYTE;
END_VAR
VAR_OUTPUT PERSISTENT
	Verified: BOOL;
	ValidCount: INT;
	InValidCount: INT;
END_VAR
VAR_OUTPUT
	WriteCount: INT;
	ReadModeActive: BOOL;
	WriteCModeActive: BOOL;
END_VAR
VAR
	//rfidHMI: ST_RFID_HMI;
	State: INT := 0;
	uRFIDInput: U_BYTE_TO_LINT;
	uRFIDDintInput: U_BYTE_TO_UDINT;
	uWriteValue: U_UINT_TO_BYTE;
	BitHeaderOutBegin: ST_BITHEADEROUT;
	BitHeaderOutEnd: ST_BITHEADEROUT;
	BitHeaderInBegin: ST_BITHEADERIN;
	BitHeaderInEnd: ST_BITHEADERIN;
	ReadFifo: FB_MyQ_UDINT;
	RdInsert: BOOL := FALSE;
	RdRemove: BOOL := FALSE;
	RdPeek: BOOL := FALSE;
	RdDump: BOOL := FALSE;
	RdReset: BOOL := FALSE;
	RdValue: UDINT := 0;
	///+++++++++++++++
	InputHeader: BYTE;
	CPRising: Tc2_Standard.R_TRIG;
	CPFalling: Tc2_Standard.F_TRIG;
	AARising: Tc2_Standard.R_TRIG;
	AAFalling: Tc2_Standard.F_TRIG;
	AERising: Tc2_Standard.R_TRIG;
	AEFalling: Tc2_Standard.F_TRIG;
	AFRising: Tc2_Standard.R_TRIG;
	AFFalling: Tc2_Standard.F_TRIG;
	TORising: Tc2_Standard.R_TRIG;
	TOFalling: Tc2_Standard.F_TRIG;
	HFRising: Tc2_Standard.R_TRIG;
	HFFalling: Tc2_Standard.F_TRIG;
	BBRising: Tc2_Standard.R_TRIG;
	BBFalling: Tc2_Standard.F_TRIG;
	OutputHeader: BYTE;
	AVRising: Tc2_Standard.R_TRIG;
	AVFalling: Tc2_Standard.F_TRIG;
	GRRising: Tc2_Standard.R_TRIG;
	GRFalling: Tc2_Standard.F_TRIG;
	KARising: Tc2_Standard.R_TRIG;
	KAFalling: Tc2_Standard.F_TRIG;
	TIRising: Tc2_Standard.R_TRIG;
	TIFalling: Tc2_Standard.F_TRIG;
	JobPendingAV: BOOL;
	GroundResetGR: BOOL;
	HeadShutdownKA: BOOL;
	ToggleTI: BOOL;
	CommandIdentifier: BYTE;
	Command: BYTE;
	CmdChangeRising: Tc2_Standard.R_TRIG;
	BeginJob: BOOL;
	ReadData: ARRAY[0..255] OF BYTE;
	WriteData: ARRAY[0..255] OF BYTE;
	JobSet: BOOL;
	JobSetRising: Tc2_Standard.R_TRIG;
	ProcessedBytes: UINT;
	RemainingBytes: UINT;
	Sequence: BYTE;
	Index: UINT;
	Length: UINT;
	tDelay: Tc2_Standard.TON;
	TOLeading: BOOL;
	TILeading: BOOL;
	CompletedSize: UINT;
	ErrorCode: BYTE;
	GroundStateReqRising: Tc2_Standard.R_TRIG;
	ShutdownReqRising: Tc2_Standard.R_TRIG;
	ReadModeRising: R_TRIG;
	uStartAddress: U_UINT_TO_BYTE;
	uNumberOfBytes: U_UINT_TO_BYTE;
	ReadRising: R_TRIG;
	ReadFalling: R_TRIG;
	WriteRising: R_TRIG;
	WriteFalling: R_TRIG;
	ReadRequest: BOOL;
	WriteRequest: BOOL;
	WriteConstant: BOOL;
	InitCRC: BOOL;
	initialized: BOOL;
	StationaryTag: BOOL;
	StationaryReadWaitCount: DINT;
	InCamWindow: BOOL;
	TagDetectedInCamWindow: BOOL;
	CamWindowFalling: F_TRIG;
	//Device: ST_Device;
END_VAR

(* This object is for Balluff BIS00LH: BIS M-400-045-001-07-S4 only *)

(*
Unless required by applicable law or agreed to in writing, software is distributed on an 
"AS IS" BASIS WITHOUT WARRANTIES OR CONDITIONS OF ANY KIND, either express or implied. 
*)


// HMI & Device setup
(*
//rfidHMI.Description:= iDevice.Description;
//rfidHMI.Symbol:= iDevice.Symbol;
//rfidHMI.Verified:= Verified;
//rfidHMI.VerifiedCount:= ValidCount;
//rfidHMI.InvalidCount:= InvalidCount;
//rfidHMI.ReadValue:= ValueRead;
//rfidHMI.DeviceReady:= DeviceReadyBB;
//rfidHMI.TagPresent:= TagPresentCP;

IF NOT initialized THEN
	rfidHMI.SizeValue:= RecipeValue;
	//rfidHMI.Cam:= Cam;
	initialized:= TRUE;
ELSIF STATUS.SIZE.NewSizeLoaded THEN
	rfidHMI.SizeValue:= RecipeValue;
	//rfidHMI.Cam:= Cam;
ELSE
	RecipeValue:= rfidHMI.SizeValue;
	//Cam:= rfidHMI.Cam;
	
END_IF
*)

ReadRising(CLK:=ReadMode AND DeviceReadyBB AND TagPresentCP AND NOT InvalidCount > 0 AND ValidCount <= NumTags);
ReadFalling(CLK:=NOT ReadMode OR InvalidCount > 0 OR ValidCount >= NumTags);
WriteRising(CLK:=WriteCMode AND DeviceReadyBB AND TagPresentCP);
WriteFalling(CLK:=NOT WriteCMode);
ReadModeRising(CLK:=ReadMode);

uStartAddress.Value:= StartAddress;
uNumberOfBytes.Value:= NumberOfBytes;

IF ReadRising.Q THEN
	ReadRequest:= TRUE;
END_IF
IF ReadFalling.Q THEN
	ReadRequest:= FALSE;
END_IF
IF WriteRising.Q AND WC_Value>0 THEN
	WriteConstant:=TRUE;
END_IF
IF WriteFalling.Q THEN
	WriteConstant:= FALSE;
END_IF

//+++++++++++++++++++++++++++++++++++++++++++
//Process Error Code
IF JobErrorAF THEN
	ErrorCode:= IO.IN.ByteArr[1];
END_IF
IF AVRising.Q THEN
	ErrorCode:=16#00;
END_IF

//Process Input Buffers
InputHeader:= IO.IN.ByteArr[0] AND IO.IN.ByteArr[9];

CPRising(CLK:=InputHeader.0);
CPFalling(CLK:=InputHeader.0);
TagPresentCP:=InputHeader.0;

AARising(CLK:=InputHeader.1);
AAFalling(CLK:=InputHeader.1);
JobAcceptedAA:=InputHeader.1;

AERising(CLK:=InputHeader.2);
AEFalling(CLK:=InputHeader.2);
JobEndAE:=InputHeader.2;

AFRising(CLK:=InputHeader.3);
AFFalling(CLK:=InputHeader.3);
JobErrorAF:=InputHeader.3;

TORising(CLK:=InputHeader.5);
TOFalling(CLK:=InputHeader.5);
ToggleTO:=InputHeader.5;

HFRising(CLK:=InputHeader.6);
HFFalling(CLK:=InputHeader.6);
HeadFailureHF:=InputHeader.6;

BBRising(CLK:=InputHeader.7);
BBFalling(CLK:=InputHeader.7);
DeviceReadyBB:=InputHeader.7;

//Process Output Buffers
IO.OUT.ByteArr[0]:=OutputHeader; IO.OUT.ByteArr[9]:=OutputHeader;

AVRising(CLK:=JobPendingAV);
AVFalling(CLK:=JobPendingAV);
OutputHeader.0:= JobPendingAV;

GRRising(CLK:=GroundResetGR);
GRFalling(CLK:=GroundResetGR);
OutputHeader.2:= GroundResetGR;

KARising(CLK:=HeadShutdownKA);
KAFalling(CLK:=HeadShutdownKA);
OutputHeader.5:= HeadShutdownKA;

TIRising(CLK:=ToggleTI);
TIFalling(CLK:=ToggleTI);
OutputHeader.6:= ToggleTI;

//Identify the command
CmdChangeRising(CLK:=ReadRequest OR WriteRequest OR InitCRC OR WriteConstant);

IF ReadRequest THEN
	CommandIdentifier:=16#01;
	Command.0:=TRUE;
END_IF
IF WriteRequest THEN
	CommandIdentifier:=16#02;
	Command.1:=TRUE;
END_IF
IF InitCRC THEN
	CommandIdentifier:=16#12;
	Command.2:=TRUE;
END_IF
IF WriteConstant THEN
	CommandIdentifier:=16#32;
	Command.3:=TRUE;
END_IF

IF CommandIdentifier = 16#01 AND ReadMode THEN
	ReadModeActive:=TRUE;
ELSE
	ReadModeActive:=FALSE;
END_IF
IF CommandIdentifier = 16#32 AND WriteCMode THEN
	WriteCModeActive:=TRUE;
ELSE
	WriteCModeActive:=FALSE;
END_IF


// Stationary vs moving tags
(*IF Cam.On <> 0 AND Cam.Off <> 0 THEN
	StationaryTag:= FALSE;
	IF Cam.On < Cam.Off THEN
		IF STATUS.MACHINE.MachinePos > Cam.On AND STATUS.MACHINE.MachinePos < Cam.Off THEN
			InCamWindow:= TRUE;
		ELSE
			InCamWindow:= FALSE;
		END_IF
	ELSE
		IF STATUS.MACHINE.MachinePos > Cam.On OR STATUS.MACHINE.MachinePos < Cam.Off THEN
			InCamWindow:= TRUE;
		ELSE
			InCamWindow:= FALSE;
		END_IF
	END_IF
ELSE
	StationaryTag:= TRUE;
END_IF
*)
StationaryTag:= TRUE;

// Stationary Tag - wait ~70 scans before reading ReadData[0]. It will not populate immediately
IF StationaryTag AND ReadMode THEN
	StationaryReadWaitCount:= StationaryReadWaitCount + 1;
ELSIF NOT ReadMode THEN
	StationaryReadWaitCount:= 0;
END_IF


// moving tag - looking for tag in cam window
IF InCamWindow AND TagPresentCP THEN
	TagDetectedInCamWindow:= TRUE;
ELSIF CamWindowFalling.Q THEN
	TagDetectedInCamWindow:= FALSE;
END_IF


//set valueread to data from RFID reader
IF (CPFalling.Q AND TagDetectedInCamWindow) OR (StationaryTag AND (StationaryReadWaitCount > 70))  THEN
	ValueRead:= ReadData[0];
	IF ValueRead = RecipeValue AND ValueRead > 0 AND ReadMode THEN
		ValidCount:= ValidCount + 1;
	END_IF
	IF ValueRead <> RecipeValue AND ReadMode THEN
		InValidCount:= InValidCount + 1;
	END_IF
	IF WriteCMode AND WC_Value > 0 THEN
		WriteCount:= WriteCount + 1;
	END_IF
END_IF
IF ValidCount = NumTags AND NumTags > 0 AND InValidCount = 0 AND ReadMode THEN
	Verified:= true;
END_IF
If ReadModeRising.Q then
	ValidCount:=0;
	InValidCount:=0;
	Verified:=FALSE;
END_IF
IF WriteRising.Q THEN
	WriteCount:= 0;
END_IF

//Load the Job
BeginJob:= CmdChangeRising.Q;

JobSetRising(CLK:=BeginJob AND NOT JobPendingAV);

IF BeginJob AND NOT JobPendingAV THEN
	IO.OUT.ByteArr[1]:= CommandIdentifier;
	IF Command.0 THEN //Read
		MEMSET(ADR(ReadData), 0, SIZEOF(ReadData));
	END_IF
	IO.OUT.ByteArr[2]:=uStartAddress.Bytes[0];
	IO.OUT.ByteArr[3]:=uStartAddress.Bytes[1];
	IO.OUT.ByteArr[4]:=uNumberOfBytes.Bytes[0];
	IO.OUT.ByteArr[5]:=uNumberOfBytes.Bytes[1];
	IF Command.3 THEN //Write Constant
		IO.OUT.ByteArr[6]:= WC_Value;
	END_IF
	ToggleTI:=FALSE;
	ProcessedBytes:=0;
	Sequence:=0;
	Index:=0;
	Length:=0;
END_IF

//Toggle AV to start the job
IF JobSetRising.Q THEN
	JobPendingAV:= TRUE;
END_IF

//Job accepted or in error clear the request
IF JobAcceptedAA THEN
	tDelay(IN:=TRUE, PT:=T#100MS);
ELSE
	tDelay(IN:=FALSE);	
END_IF
IF JobAcceptedAA OR JobErrorAF THEN
	ReadRequest:=FALSE;
	WriteRequest:=FALSE;
	InitCRC:=FALSE;
	WriteConstant:=FALSE;	
END_IF

//compute how many bytes remaining
RemainingBytes:=NumberOfBytes-ProcessedBytes;

//Compute necessary length of the next read/write cycle
IF RemainingBytes > 8 THEN
	Length:=8;
END_IF
IF RemainingBytes <=8 THEN
	Length:=RemainingBytes;
END_IF

//Create the index that evaluates the start address of the next read/write cycle
Index:= NumberOfBytes-RemainingBytes;
IF Index > 255 THEN
	Index:=255;
END_IF

IF tDelay.Q AND NOT TOLeading AND NOT TILeading THEN
	IF ToggleTO THEN
		TOLeading:=TRUE;
	END_IF
	IF NOT ToggleTO THEN
		TILeading:=TRUE;
	END_IF
END_IF

IF TORising.Q THEN
	Sequence.0:=TRUE;
END_IF
IF TOFalling.Q THEN
	Sequence.1:=TRUE;
END_IF

//Once the job is accepted and TI is low or on lo-hi/hi-lo transition of TO, copy the data
IF (Sequence.0 OR Sequence.1 OR (TILeading AND Index = 0)) AND NOT Sequence.2 THEN
	IF Command.0 AND JobEndAE THEN
		MEMCPY(ADR(ReadData[Index]), ADR(IO.IN.ByteArr[1]), Length);
		Sequence.2:= TRUE;
	END_IF
	IF Command.1 AND tDelay.Q THEN
		MEMCPY(ADR(IO.OUT.ByteArr[1]), ADR(WriteData[Index]), Length);
		Sequence.2:= TRUE;
	END_IF
	ProcessedBytes:= Length+ProcessedBytes;
END_IF

IF Sequence.2 THEN
	IF TOLeading THEN
		IF Sequence.0 THEN
			ToggleTI:=TRUE;
			Sequence.0:=FALSE;
			Sequence.3:=TRUE;
		END_IF
		IF Sequence.1 THEN
			ToggleTI:=FALSE;
			Sequence.1:=FALSE;
			Sequence.3:=TRUE;
		END_IF
	END_IF
	IF TILeading THEN
		IF Sequence.0 THEN
			ToggleTI:=FALSE;
			Sequence.0:=FALSE;
			Sequence.3:=TRUE;
		END_IF
		IF Sequence.1 OR Index = 0 THEN
			ToggleTI:=TRUE;
			Sequence.1:=FALSE;
			Sequence.3:=TRUE;
		END_IF
	END_IF
END_IF

IF Sequence.3 THEN
	Sequence.2:=FALSE;
END_IF

//On the falling edge of the AA bit, transition TI low, compute the size of the operation completed, and clear the working data
IF (Command.0 AND RemainingBytes = 0) OR (Command.1 OR Command.2 OR Command.3 AND JobEndAE) OR AFRising.Q OR GroundResetGR THEN
	JobPendingAV:=FALSE;
	ToggleTI:=FALSE;
	CompletedSize:=ProcessedBytes;
	ProcessedBytes:=0;
	Sequence:=0;
	Command:=0;
	Index:=0;
	RemainingBytes:=0;
	Length:=0;
END_IF

//Reset After Job Complete
IF AAFalling.Q THEN
	CompletedSize:=ProcessedBytes;
	ProcessedBytes:=0;
	Sequence:=0;
	Command:=0;
	TOLeading:=FALSE;
	TILeading:=FALSE;
	ToggleTI:=FALSE;
END_IF

//Process Ground State Request
GroundStateReqRising(CLK:=GroundStateRequest AND NOT ShutdownRequest);
IF GroundStateReqRising.Q THEN
	GroundResetGR:=TRUE;
END_IF
IF GroundResetGR AND NOT DeviceReadyBB AND NOT GroundStateRequest THEN
	GroundResetGR:=FALSE;
END_IF
 
//Process Head Shutdown Request
ShutdownReqRising(CLK:=ShutdownRequest AND NOT GroundStateRequest);
IF ShutdownReqRising.Q THEN
	HeadShutdownKA:=TRUE;
END_IF
IF HeadShutdownKA AND HeadFailureHF AND NOT ShutdownRequest THEN
	HeadShutdownKA:=FALSE;
END_IF

(*
Device.Desc:= iDevice.Description;
Device.Symbol:= iDevice.Symbol;

CamWindowFalling(CLK:=InCamWindow);

ABORT_MissingTag(
	Trigger:= NOT StationaryTag AND CamWindowFalling.Q AND NOT TagDetectedInCamWindow AND ReadModeActive, 
	Reset:= STATUS.MACHINE.PrepareToStartPulse, 
	Code:= 0, 
	Message:= 'Missing RFID Tag', 
	Device:= Device, 
	Location:= iDevice.Location, 
	Active=> );
	
ABORT_WrongTag(
	Trigger:= ReadModeActive AND CPFalling.Q AND ValueRead <> RecipeValue, 
	Reset:= STATUS.MACHINE.PrepareToStartPulse, 
	Code:= 0, 
	Message:= 'Wrong RFID Tag', 
	Device:= Device, 
	Location:= iDevice.Location, 
	Active=> );

	
// this will only occur during read mode, reset counters when not a good read
IF ABORT_MissingTag.Active OR ABORT_WrongTag.Active THEN
	ValidCount:= 0;
	InValidCount:= 0;
END_IF
*)

END_FUNCTION_BLOCK

// ---- Application/CSP/Main/Services/RFID FB/FB_MyQ_UDINT.TcPOU
FUNCTION_BLOCK FB_MyQ_UDINT
VAR_INPUT
	/// NewValue : the value of the new data inserted into the queue 
	NewValue: UDINT;
END_VAR
VAR_IN_OUT
	/// LoadNew : triggers loading of NewValue 
	Insert: BOOL;
	/// GetOld	: retrieve the oldest value in the queue 
	Remove: BOOL;
	/// Peek		: View but do not retrieve the oldest value in the queue, queue is not affected 
	Peek: BOOL;
	Dump: BOOL;
	/// Reset	: Zero out all counters and queues 
	Reset: BOOL;
END_VAR
VAR_OUTPUT
	/// OldValue	: the oldest value retrieved from the queue when the 'GetOld' input is triggered 
	OldValue: UDINT;
	/// PeekValue : the oldest value viewed but not retrieved (queue is not affected) from the queue when 'Peek' input is triggered 
	PeekValue: UDINT;
	FifoDump: ARRAY[1..QUEUESIZE] OF UDINT;
	FifoSize: INT;
	/// Count	: number of values in the queue 
	Count: INT;
	/// ExecutionCntr	: number of times this function block has been called 
	ExecutionCntr: DINT;
END_VAR
VAR CONSTANT
	QUEUESIZE: INT := 12;
END_VAR
VAR
	HoldQueue: ARRAY[1..QUEUESIZE] OF UDINT;
	rtInsert: R_TRIG;
	rtRemove: R_TRIG;
	rtPeek: R_TRIG;
	rtDump: R_TRIG;
	rtReset: R_TRIG;
	i: INT;
	ProcessQueue: ARRAY[1..QUEUESIZE] OF UDINT;
	Elements: INT;
END_VAR

rtInsert(CLK:=Insert);
rtRemove(CLK:=Remove);
rtPeek(CLK:=Peek);
rtDump(CLK:=Dump);
rtReset(CLK:=Reset);

IF rtInsert.Q THEN
	IF Elements < QUEUESIZE THEN
		Elements := Elements + 1;
		ProcessQueue[Elements]:= NewValue;
	ELSE
		Elements := QUEUESIZE;
		ProcessQueue[Elements]:= NewValue;	
	END_IF
	Insert:=FALSE;
END_IF

IF rtRemove.Q THEN
	IF Elements > 0 THEN
		OldValue := ProcessQueue[1];
		FOR i:= 1 TO QUEUESIZE DO
			HoldQueue[i] := ProcessQueue[i];	
		END_FOR
		FOR i:= 1 TO QUEUESIZE-1 DO
			ProcessQueue[i] := HoldQueue[i+1];	
		END_FOR
		Elements := Elements - 1;
	END_IF
	Remove:=FALSE;
END_IF

IF rtPeek.Q THEN
	IF Elements > 0 THEN
		PeekValue := ProcessQueue[1];
	END_IF
	Peek:=FALSE;
END_IF

IF rtDump.Q THEN
	FifoDump := ProcessQueue;
	Dump:=FALSE;
END_IF

IF rtReset.Q THEN
	FOR i:= 1 TO QUEUESIZE DO
		HoldQueue[i] := 0;
		ProcessQueue[i] := 0;
		FifoDump[i] := 0;	
	END_FOR
	Elements := 0;
	ExecutionCntr:= 0;
	Reset:=FALSE;
END_IF

Count := Elements;
ExecutionCntr:= ExecutionCntr+1;
FifoSize:= QUEUESIZE;

END_FUNCTION_BLOCK

// ---- Application/CSP/Main/Services/RFID FB/IO_RFID.TcPOU
FUNCTION_BLOCK IO_RFID
VAR_INPUT
	BitHeader1Out AT %Q*: BYTE;
	Byte1OutCmdDesig_Data AT %Q*: BYTE;
	Byte2OutStartAddrLow_Data AT %Q*: BYTE;
	Byte3OutStartAddrHigh_Data AT %Q*: BYTE;
	Byte4OutNumBytesLow_Data AT %Q*: BYTE;
	Byte5OutNumBytesHigh_Data AT %Q*: BYTE;
	Byte6OutData AT %Q*: BYTE;
	Byte7OutData AT %Q*: BYTE;
	Byte8OutData AT %Q*: BYTE;
	BitHeader2Out AT %Q*: BYTE;
	OutputByteArr AT %Q*: ARRAY[0..9] OF BYTE;
END_VAR
VAR_OUTPUT
	DeviceDiag AT %I*: BOOL;
	DeviceState AT %I*: BOOL;
	ChannelState AT %I*: USINT;
	InfoDataState AT %I*: UINT;
	BitHeader1In AT %I*: BYTE;
	Byte1InErrCode_Data_HighVer AT %I*: BYTE;
	Byte2InData_LowVer AT %I*: BYTE;
	Byte3InData AT %I*: BYTE;
	Byte4InData AT %I*: BYTE;
	Byte5InData AT %I*: BYTE;
	Byte6InData AT %I*: BYTE;
	Byte7InData AT %I*: BYTE;
	Byte8InData AT %I*: BYTE;
	BitHeader2In AT %I*: BYTE;
	InputByteArr AT %I*: ARRAY[0..9] OF BYTE;
END_VAR

END_FUNCTION_BLOCK

// ---- Application/CSP/Main/Services/RFID FB/RFID_FB.TcPOU
PROGRAM RFID_FB
VAR
	RFID_FB:							FB_BIS00LH;
	RFID_IO:							ST_BIS00LH_IO;	

END_VAR

RFID_FB(IO := RFID_IO);

END_PROGRAM

// ---- Application/CSP/Transfer/Main/csp_transfer_main.TcPOU
(*********************************** G.D S.p.A. - Technical Department ***********************************
============= PROGRAM INFO ============
FOLDER:             TBD
MACHINES INVOLVED:  TBD 

============= DESCRIPTION =============
csp main program

============= REVISIONS ===============
Date		Version	 	Author      	Description             
----------	-------		------------  	--------------------------------------------
2019/04/05 	0000.00	 	M.Grasso		Creation of the PRG

**********************************************************************************************************)
(*$R
	process_ref := prc;
$*)
PROGRAM csp_transfer_main
VAR
	prc:												process;
	prc_path:											STRING;
	
	temperature_fault_di:								digital_input;
	temperature_fault_dchk:								digital_check;
	
END_VAR

VAR_INPUT
	i_cabinet_is_running:								BOOL;
	
END_VAR

VAR_OUTPUT
	o_reset_button:										BOOL;
	o_start_button:										BOOL;
END_VAR

_read_var_input();

_object_manager();

IF NOT objects_running()
THEN
	RETURN;	
END_IF

_read_process_image();

_mode_manager();

CASE process_get_mode(prc) of
	MODE_ABSENT,
	MODE_INACTIVE:
		RETURN;
	MODE_TEST:
		_handle_process_test();
END_CASE

_set_runtime_properties();

(********************************* BODY *********************************)




(************************************************************************)

_handle_messages();

_write_output();

ACTION _handle_messages:
;
END_ACTION

ACTION _handle_process_test:
;
END_ACTION

ACTION _mode_manager:
IF process_mode_req_is_pending(prc)
THEN
    process_apply_mode_req_first_step(prc);
    CASE process_get_mode(prc) OF
        MODE_TO_ABSENT:
			;
        MODE_TO_INACTIVE:
			;
        MODE_TO_TEST:
			;
        MODE_TO_OPERATIONAL:
			;
    END_CASE
    process_apply_mode_req_second_step(prc);
END_IF
END_ACTION

ACTION _object_manager:
IF objects_initialization()
THEN
	sub_process_init(
		object_name					:= 'csp_transfer_main.prc', 
		process						:= csp_transfer.prc, 
		CONVERSION_this				:= prc);
		
	prc_path 						:= process_get_path(prc);
	
	
	digital_input_init(
		object_name					:= CONCAT(prc_path, '_temperature_fault_di'), 
		polarity_direct				:= TRUE, 
		process						:= prc, 
		CONVERSION_this				:= temperature_fault_di);
		
	digital_check_init(
		object_name					:= CONCAT(prc_path, '_temperature_fault_dchk'),
		alarm_if_input_off			:= FALSE,
		alarm_delay					:= 1000,
		enabled_at_powerup			:= TRUE,
		process						:= prc,
		CONVERSION_this				:= temperature_fault_dchk);

	digital_check_add_di(
		di							:= temperature_fault_di,
		CONVERSION_this				:= temperature_fault_dchk);
		
END_IF

IF objects_running()
THEN
	process_cycle(prc);
	digital_check_cycle(temperature_fault_dchk);
END_IF
END_ACTION

ACTION _read_process_image:
;
END_ACTION

ACTION _read_var_input:
//i_cabinet_is_running					:= cb.o_machine_is_running; (*MARCO*)
//i_machine_motor_axis_ref				:= ADR(csp_main_motorization_virtualManager.virtual_master_test); //TODO: this will need an update
(*
i_carton_closing_shift_is_empty			:= csp_cartonClosing_shiftRegister.is_empty;
i_carton_filling_shift_is_empty			:= wu_cartonFilling_shiftRegister.is_empty;
i_carton_forming_shift_is_empty			:= wu_cartonForming_shiftRegister.is_empty;
i_carton_pickup_shift_is_empty			:= wu_cartonPickup_shiftRegister.is_empty;
i_cups_feeding_shift_is_empty			:= wu_cupsFeeding_shiftRegister.is_empty;
i_exit_shift_is_empty					:= wu_exit_shiftRegister.is_empty;
i_twisted_cups_shift_is_empty			:= wu_twistedCups_shiftRegister.is_empty;

i_machine_motor_axis_ref				:= ADR(wu_cartonForming_motorization.axis);
i_drums_motor_axis_ref					:= ADR(wu_cartonPickup_drums_motorization.axis);

i_R1_robot_source_shift_ref				:= ADR(wu_cupsFeeding_shiftRegister.outer_sr); 
i_R2_robot_source_shift_ref				:= ADR(wu_cupsFeeding_shiftRegister.inner_sr);

i_twisted_cups_inner_shift_ref			:= ADR(wu_twistedCups_shiftRegister.inner_sr);
i_twisted_cups_outer_shift_ref			:= ADR(wu_twistedCups_shiftRegister.outer_sr);

i_carton_filling_shift_ref				:= ADR(wu_cartonFilling_shiftRegister.sr);
*)
END_ACTION

ACTION _set_runtime_properties:
;
END_ACTION

ACTION _write_output:
o_reset_button	:= csp_transfer_main_services_pushbuttons.reset_pressed;
o_start_button	:= csp_transfer_main_services_pushbuttons.start_pressed;
END_ACTION

END_PROGRAM

// ---- POUs/AFL extensions/analog_actuator/analog_actuator_cycle.TcPOU
(*$
	Handles the state machine of the object, has to be called once per task cycle <br/>
	<p>
	Against certain errors the cpu can be stopped at the first cycle of the caller task, <br/> 
	in this case the cause can be inspected in the global struct <i>framework.abort_error</i>: <br/>
	<br/>
	<li> <b>ERRORID_1 = 17</b>: Active digital_input not added. </li>
	<li> <b>ERRORID_1 = 19</b>: Inactive digital_input not added. </li>
	</p>

$*)
FUNCTION analog_actuator_cycle : VOID

VAR_IN_OUT
    CONVERSION_this:	analog_actuator;	(*$ Instance to which the method applies $*)
END_VAR

IF NOT CONVERSION_this.CONVERSION_private.cycle_is_active
THEN
	descriptor_set_task_id(CONVERSION_this.descriptor);

	IF analog_actuator_is_not_initialized(CONVERSION_this)
	THEN
		framework_object_not_initialized_get_name(
			object_address := ADR(CONVERSION_this),
			object_size := SIZEOF(CONVERSION_this),
			abort := TRUE,
			error_str_1 := 'object not initialized',
			error_str_2 := ''
		);
	    RETURN;
	END_IF

	CONVERSION_this.CONVERSION_private.cycle_is_active := TRUE;
END_IF

IF descriptor_mode_req_is_pending(CONVERSION_this.descriptor) THEN
    analog_actuator_change_mode(CONVERSION_this);
END_IF

IF CONVERSION_this.has_di_ready
THEN
	digital_check_cycle(CONVERSION_this.ready_dchk);
END_IF

IF CONVERSION_this.has_di_active
THEN
	digital_check_cycle(CONVERSION_this.active_dchk);
	digital_check_cycle(CONVERSION_this.inactive_dchk);
END_IF

IF CONVERSION_this.has_ai_feedback
THEN
	analog_check_cycle(CONVERSION_this.feedback_achk);
END_IF

CASE descriptor_get_mode(CONVERSION_this.descriptor) OF
	MODE_ABSENT:
		RETURN;

	MODE_TO_INACTIVE:
		;		(*$FIXME: To inactive mode strategy to handle. $*)

	MODE_INACTIVE:
		;		(*$FIXME: Inactive mode to handle. $*)

	MODE_TEST:
		CONVERSION_this.command := analog_actuator_test_command_handler(CONVERSION_this);

	MODE_OPERATIONAL:
		CONVERSION_this.command := CONVERSION_this.operational_command;

END_CASE;

analog_actuator_read_inputs(CONVERSION_this);
analog_actuator_submit_command(CONVERSION_this);

CONVERSION_this.ao_setpoint_value := CONVERSION_this.analog_physical_command;

IF CONVERSION_this.has_ai_feedback
THEN
	CONVERSION_this.ai_feedback_value := analog_input_physical_read(CONVERSION_this.ai_feedback^);
ELSE
	CONVERSION_this.ai_feedback_value := 0;
END_IF

(*transition states*)
CASE CONVERSION_this.status OF
	ANALOG_ACTUATOR_STATUS_INIT:
    	CONVERSION_this.status := ANALOG_ACTUATOR_STATUS_INACTIVE;

    ANALOG_ACTUATOR_STATUS_ACTIVATING:
		IF CONVERSION_this.is_active AND NOT CONVERSION_this.is_inactive
		THEN
			(*TEST EV*)
			IF	descriptor_get_mode(CONVERSION_this.descriptor) = MODE_OPERATIONAL
			THEN
				CONVERSION_this.operational_command := ANALOG_ACTUATOR_CMD_NONE;
			END_IF

			IF	descriptor_get_mode(CONVERSION_this.descriptor) = MODE_TEST
			THEN
				CONVERSION_this.test.command := ANALOG_ACTUATOR_TEST_CMD_IDLE;
			END_IF

			IF CONVERSION_this.has_ai_feedback
			THEN
				analog_check_set_min_value(CONVERSION_this.analog_physical_command - CONVERSION_this.feedback_lower_tolerance, CONVERSION_this.feedback_achk);
				analog_check_set_max_value(CONVERSION_this.analog_physical_command + CONVERSION_this.feedback_upper_tolerance, CONVERSION_this.feedback_achk);
				analog_check_enable(CONVERSION_this.feedback_achk);
			END_IF

			CONVERSION_this.command := ANALOG_ACTUATOR_CMD_NONE;
			CONVERSION_this.status := ANALOG_ACTUATOR_STATUS_ACTIVE;
		ELSE
			IF CONVERSION_this.has_ai_feedback
			THEN
				analog_check_disable(CONVERSION_this.feedback_achk);
			END_IF
		END_IF
		IF descriptor_is_ready(CONVERSION_this.descriptor)
		THEN
			CONVERSION_this.active_elapsed_time := timer_get_elapsed_time(CONVERSION_this.timer);
		END_IF


    ANALOG_ACTUATOR_STATUS_DEACTIVATING:
        IF CONVERSION_this.is_inactive AND NOT CONVERSION_this.is_active
		THEN
			(*TEST EV*)
			IF	descriptor_get_mode(CONVERSION_this.descriptor) = MODE_OPERATIONAL
			THEN
				CONVERSION_this.operational_command := ANALOG_ACTUATOR_CMD_NONE;
			END_IF

			IF	descriptor_get_mode(CONVERSION_this.descriptor) = MODE_TEST
			THEN
				CONVERSION_this.test.command := ANALOG_ACTUATOR_TEST_CMD_IDLE;
			END_IF

			IF CONVERSION_this.has_ai_feedback
			THEN
				analog_check_disable(CONVERSION_this.feedback_achk);
			END_IF

			CONVERSION_this.command := ANALOG_ACTUATOR_CMD_NONE;
			CONVERSION_this.status := ANALOG_ACTUATOR_STATUS_INACTIVE;
		END_IF

		IF CONVERSION_this.has_ai_feedback
		THEN
			analog_check_disable(CONVERSION_this.feedback_achk);
		END_IF

		IF descriptor_is_ready(CONVERSION_this.descriptor)
		THEN
			CONVERSION_this.deactive_elapsed_time := timer_get_elapsed_time(CONVERSION_this.timer);
		END_IF

    ANALOG_ACTUATOR_STATUS_FAULTED:
       CASE CONVERSION_this.fault_reaction OF
			ANALOG_ACTUATOR_FAULT_REACTION_DEACTIVATING:
				analog_output_physical_write(physical_value := 0, CONVERSION_this := CONVERSION_this.ao_setpoint^);	(*todo: to consider also percent write*)
				IF CONVERSION_this.has_do_activate
				THEN
					digital_output_reset(CONVERSION_this.do_activate^);
				END_IF
				CONVERSION_this.operational_command := ANALOG_ACTUATOR_CMD_DEACTIVATE;
				CONVERSION_this.test.command := ANALOG_ACTUATOR_TEST_CMD_DEACTIVATE;

			ANALOG_ACTUATOR_FAULT_REACTION_HOLD,
			ANALOG_ACTUATOR_FAULT_REACTION_IGNORE:
				CONVERSION_this.operational_command := ANALOG_ACTUATOR_CMD_NONE;
				CONVERSION_this.test.command := ANALOG_ACTUATOR_TEST_CMD_IDLE;
		END_CASE;

		IF CONVERSION_this.has_ai_feedback
		THEN
			analog_check_disable(CONVERSION_this.feedback_achk);
		END_IF

END_CASE;

(*dynamic diagnosis*)
CASE CONVERSION_this.status OF

    ANALOG_ACTUATOR_STATUS_ACTIVATING:

        IF timer_is_expired(CONVERSION_this.timer)
        THEN
			IF 	CONVERSION_this.has_ai_feedback
				OR
				CONVERSION_this.has_di_active
			THEN
				analog_actuator_set_snapshot(
					errorID_1 := 10,
					errorID_2 := 0,
					errorID_3 := 0,
					CONVERSION_this := CONVERSION_this.active_fem
					);

				IF CONVERSION_this.fault_reaction <> ANALOG_ACTUATOR_FAULT_REACTION_IGNORE
				THEN
					CONVERSION_this.status := ANALOG_ACTUATOR_STATUS_FAULTED;
				END_IF
			END_IF
		END_IF

	ANALOG_ACTUATOR_STATUS_INACTIVE:

		IF CONVERSION_this.has_di_active
		THEN
			digital_check_enable(CONVERSION_this.inactive_dchk);
		END_IF

    ANALOG_ACTUATOR_STATUS_DEACTIVATING:

        IF timer_is_expired(CONVERSION_this.timer)
        THEN
			IF 	CONVERSION_this.has_ai_feedback
				OR
				CONVERSION_this.has_di_active
			THEN
				analog_actuator_set_snapshot(
					errorID_1 := 11,
					errorID_2 := 0,
					errorID_3 := 0,
					CONVERSION_this := CONVERSION_this.inactive_fem
					);

				IF CONVERSION_this.fault_reaction <> ANALOG_ACTUATOR_FAULT_REACTION_IGNORE
				THEN
					CONVERSION_this.status := ANALOG_ACTUATOR_STATUS_FAULTED;
				END_IF
			END_IF
		END_IF
END_CASE;

(*static diagnosis*)
IF 	CONVERSION_this.has_di_ready
THEN
	digital_check_enable(CONVERSION_this.ready_dchk);
	IF message_is_on(CONVERSION_this.ready_dchk.alarm_asm.message)
	THEN
		IF CONVERSION_this.fault_reaction <> ANALOG_ACTUATOR_FAULT_REACTION_IGNORE
		THEN
			CONVERSION_this.status := ANALOG_ACTUATOR_STATUS_FAULTED;
		END_IF
	END_IF
END_IF

IF 	CONVERSION_this.has_di_active
THEN
	IF	CONVERSION_this.status = ANALOG_ACTUATOR_STATUS_ACTIVE
	THEN
		digital_check_enable(CONVERSION_this.active_dchk);
		IF message_is_on(CONVERSION_this.active_dchk.alarm_asm.message)
		THEN
			IF CONVERSION_this.fault_reaction <> ANALOG_ACTUATOR_FAULT_REACTION_IGNORE
			THEN
				CONVERSION_this.status := ANALOG_ACTUATOR_STATUS_FAULTED;
			END_IF
		END_IF
	ELSE
		digital_check_disable(CONVERSION_this.active_dchk);
	END_IF
END_IF

IF 	CONVERSION_this.has_di_active
THEN
	IF	CONVERSION_this.status = ANALOG_ACTUATOR_STATUS_INACTIVE
	THEN
		digital_check_enable(CONVERSION_this.inactive_dchk);
		IF message_is_on(CONVERSION_this.inactive_dchk.alarm_asm.message)
		THEN
			IF CONVERSION_this.fault_reaction <> ANALOG_ACTUATOR_FAULT_REACTION_IGNORE
			THEN
				CONVERSION_this.status := ANALOG_ACTUATOR_STATUS_FAULTED;
			END_IF
		END_IF
	ELSE
		digital_check_disable(CONVERSION_this.inactive_dchk);
	END_IF
END_IF

(*fault manager*)
CASE descriptor_get_stop_status(CONVERSION_this.descriptor) OF
    STOP_GOING_ON:
		descriptor_apply_stop(CONVERSION_this.descriptor);
    STOP_ON:
		IF descriptor_get_reset_level(CONVERSION_this.descriptor)
        THEN
            CONVERSION_this.status := ANALOG_ACTUATOR_STATUS_INIT;
			CONVERSION_this.command := CONVERSION_this.operational_command;
			analog_actuator_submit_command(CONVERSION_this);
        END_IF
	STOP_OFF:
		IF 	CONVERSION_this.status
			=
			ANALOG_ACTUATOR_STATUS_FAULTED
		THEN
			IF descriptor_get_reset_level(CONVERSION_this.descriptor)
	        THEN
	            CONVERSION_this.status := ANALOG_ACTUATOR_STATUS_INIT;
				CONVERSION_this.command := CONVERSION_this.operational_command;
				analog_actuator_submit_command(CONVERSION_this);
	        END_IF
		END_IF
END_CASE;

END_FUNCTION

// ---- POUs/AFL extensions/analog_actuator/private/analog_actuator_is_not_initialized.TcPOU
(* Function that returns if an object is not initialized. *)
FUNCTION analog_actuator_is_not_initialized : BOOL
VAR_IN_OUT
	CONVERSION_this:	analog_actuator;	(* object reference *)
END_VAR

analog_actuator_is_not_initialized:=NOT CONVERSION_this.CONVERSION_private.initialized;

END_FUNCTION

// ---- POUs/AFL extensions/analog_actuator/private/analog_actuator_change_mode.TcPOU
(* Function that allows to change the analog_actuator mode. <br/>
	(ACTIVE, INACTIVE, ABSENT etc.....) *)
FUNCTION analog_actuator_change_mode : VOID

VAR
	i:		DINT;
END_VAR
(*All VAR_IN_OUT variables have been moved to the end of the declaration due to compatibility reasons*)
VAR_IN_OUT
    CONVERSION_this:	analog_actuator;
END_VAR

descriptor_apply_mode_req_first_step(CONVERSION_this.descriptor);

IF  descriptor_get_mode(CONVERSION_this.descriptor) = MODE_TO_ABSENT
    OR
    descriptor_get_mode(CONVERSION_this.descriptor) = MODE_TO_INACTIVE
    OR
    descriptor_get_mode(CONVERSION_this.descriptor) = MODE_TO_OPERATIONAL
    OR
    descriptor_get_mode(CONVERSION_this.descriptor) = MODE_TO_TEST
THEN
	CONVERSION_this.status := ANALOG_ACTUATOR_STATUS_INIT;
	CONVERSION_this.operational_command := ANALOG_ACTUATOR_CMD_NONE;
	IF CONVERSION_this.has_do_activate
	THEN
		digital_output_reset(CONVERSION_this.do_activate^);
	END_IF
	analog_output_physical_write(physical_value := 0, CONVERSION_this := CONVERSION_this.ao_setpoint^);
END_IF

IF 	CONVERSION_this.light_test_active = TRUE
	AND
	descriptor_get_mode(CONVERSION_this.descriptor) = MODE_TO_TEST
THEN
	IF	analog_actuator_is_active(CONVERSION_this)
	THEN
		CONVERSION_this.operational_command := ANALOG_ACTUATOR_CMD_ACTIVATE;
	END_IF

	IF	analog_actuator_is_inactive(CONVERSION_this)
	THEN
		CONVERSION_this.operational_command := ANALOG_ACTUATOR_CMD_DEACTIVATE;
	END_IF

END_IF

IF  descriptor_get_mode(CONVERSION_this.descriptor) <> MODE_TO_OPERATIONAL
	AND
	descriptor_get_mode(CONVERSION_this.descriptor) <> MODE_TO_TEST
THEN
	CONVERSION_this.operational_command := ANALOG_ACTUATOR_CMD_NONE;
END_IF


CONVERSION_this.test.command := ANALOG_ACTUATOR_TEST_CMD_IDLE;
CONVERSION_this.command := ANALOG_ACTUATOR_CMD_NONE;

FOR i := 0 TO ANALOG_ACTUATOR_MAX_TEST_COMMANDS
DO
	CONVERSION_this.test.command_info[i].available := FALSE;
	CONVERSION_this.test.command_info[i].status := TEST_COMMAND_STATUS_NOT_DONE;
END_FOR

descriptor_apply_mode_req_second_step(CONVERSION_this.descriptor);

END_FUNCTION

// ---- POUs/AFL extensions/analog_actuator/status/analog_actuator_is_active.TcPOU
(*$
	Returns <i>TRUE</i> if the status of the instance <b><i>this</i></b> is
	<a href="#analog_actuator_status_enum"><i>ANALOG_ACTUATOR_STATUS_ACTIVE</i></a>, 
	<i>FALSE</i> otherwise.
$*)
FUNCTION analog_actuator_is_active : BOOL
VAR_IN_OUT
    CONVERSION_this:	analog_actuator;	(*$ Instance to which the method applies $*)
END_VAR

analog_actuator_is_active := (CONVERSION_this.status = ANALOG_ACTUATOR_STATUS_ACTIVE);

END_FUNCTION

// ---- POUs/AFL extensions/analog_actuator/status/analog_actuator_is_inactive.TcPOU
(*$
	Returns <i>TRUE</i> if the status of the instance <b><i>this</i></b> is
	<a href="#analog_actuator_status_enum"><i>ANALOG_ACTUATOR_STATUS_INACTIVE</i></a>, 
	<i>FALSE</i> otherwise.
$*)
FUNCTION analog_actuator_is_inactive: BOOL
VAR_IN_OUT
    CONVERSION_this:	analog_actuator;	(*$ Instance to which the method applies $*)
END_VAR

IF descriptor_get_mode(CONVERSION_this.descriptor) = MODE_ABSENT
THEN
	analog_actuator_is_inactive := TRUE;
	RETURN;
END_IF

analog_actuator_is_inactive := (CONVERSION_this.status = ANALOG_ACTUATOR_STATUS_INACTIVE);

END_FUNCTION

// ---- POUs/AFL extensions/analog_actuator/private/analog_actuator_test_command_handler.TcPOU
FUNCTION analog_actuator_test_command_handler : analog_actuator_command_enum
VAR_IN_OUT
    CONVERSION_this:	analog_actuator;	(* Instance to which the method applies *)
END_VAR

analog_actuator_test_command_handler := ANALOG_ACTUATOR_CMD_NONE;
IF descriptor_is_ready(CONVERSION_this.descriptor)
THEN
	(*Test command info handling*)
	IF	CONVERSION_this.status <> ANALOG_ACTUATOR_STATUS_FAULTED
	THEN
	    CONVERSION_this.test.command_info[ANALOG_ACTUATOR_TEST_CMD_ACTIVATE].available := TRUE;
	ELSE
	    CONVERSION_this.test.command_info[ANALOG_ACTUATOR_TEST_CMD_ACTIVATE].available := FALSE;
	END_IF
	IF  CONVERSION_this.status = ANALOG_ACTUATOR_STATUS_ACTIVATING
	THEN
	    CONVERSION_this.test.command_info[ANALOG_ACTUATOR_TEST_CMD_ACTIVATE].status := TEST_COMMAND_STATUS_RUNNING;
	ELSIF CONVERSION_this.status = ANALOG_ACTUATOR_STATUS_ACTIVE
	THEN
		CONVERSION_this.test.command_info[ANALOG_ACTUATOR_TEST_CMD_ACTIVATE].status := TEST_COMMAND_STATUS_DONE;
	ELSE
		CONVERSION_this.test.command_info[ANALOG_ACTUATOR_TEST_CMD_ACTIVATE].status := TEST_COMMAND_STATUS_NOT_DONE;
	END_IF

	IF	CONVERSION_this.status = ANALOG_ACTUATOR_STATUS_ACTIVE
	THEN
	    CONVERSION_this.test.command_info[ANALOG_ACTUATOR_TEST_CMD_DEACTIVATE].available := TRUE;
	ELSE
	    CONVERSION_this.test.command_info[ANALOG_ACTUATOR_TEST_CMD_DEACTIVATE].available := FALSE;
	END_IF
	IF  CONVERSION_this.status = ANALOG_ACTUATOR_STATUS_DEACTIVATING
	THEN
	    CONVERSION_this.test.command_info[ANALOG_ACTUATOR_TEST_CMD_DEACTIVATE].status := TEST_COMMAND_STATUS_RUNNING;
	ELSIF CONVERSION_this.status = ANALOG_ACTUATOR_STATUS_INACTIVE
	THEN
		CONVERSION_this.test.command_info[ANALOG_ACTUATOR_TEST_CMD_DEACTIVATE].status := TEST_COMMAND_STATUS_DONE;
	ELSE
		CONVERSION_this.test.command_info[ANALOG_ACTUATOR_TEST_CMD_DEACTIVATE].status := TEST_COMMAND_STATUS_NOT_DONE;
	END_IF
	IF	CONVERSION_this.status = ANALOG_ACTUATOR_STATUS_INIT
	THEN
	    CONVERSION_this.test.command_info[ANALOG_ACTUATOR_TEST_CMD_ACTIVATE].available := TRUE;
		CONVERSION_this.test.command_info[ANALOG_ACTUATOR_TEST_CMD_DEACTIVATE].available := TRUE;
		CONVERSION_this.test.command_info[ANALOG_ACTUATOR_TEST_CMD_ACTIVATE].status := TEST_COMMAND_STATUS_NOT_DONE;
		CONVERSION_this.test.command_info[ANALOG_ACTUATOR_TEST_CMD_DEACTIVATE].status := TEST_COMMAND_STATUS_NOT_DONE;
	END_IF

	(*Enumerative convertion from analog_actuator_test_command_enum to analog_actuator_command_enum *)
	CASE CONVERSION_this.test.command OF
		ANALOG_ACTUATOR_TEST_CMD_ACTIVATE:
		IF CONVERSION_this.test.command_info[ANALOG_ACTUATOR_TEST_CMD_ACTIVATE].available
		THEN
			CONVERSION_this.analog_physical_command := CONVERSION_this.test.physical_value;
			analog_actuator_test_command_handler := ANALOG_ACTUATOR_CMD_ACTIVATE;
		END_IF

		ANALOG_ACTUATOR_TEST_CMD_DEACTIVATE:
		IF CONVERSION_this.test.command_info[ANALOG_ACTUATOR_TEST_CMD_DEACTIVATE].available
		THEN
			CONVERSION_this.analog_physical_command := 0;
			analog_actuator_test_command_handler := ANALOG_ACTUATOR_CMD_DEACTIVATE;
		END_IF
	END_CASE
END_IF

END_FUNCTION

// ---- POUs/AFL extensions/analog_actuator/private/analog_actuator_read_inputs.TcPOU
(* Function that updates the feedback sensors states of the
	analog_actuator specified by the parameter 'this'. *)
FUNCTION analog_actuator_read_inputs : VOID
VAR
	input_active: BOOL;
END_VAR
VAR_IN_OUT
    CONVERSION_this:		analog_actuator;	(*$ analog_actuator reference $*)
END_VAR

IF CONVERSION_this.has_di_active
THEN
	input_active := digital_input_is_active(CONVERSION_this.di_active^);
ELSE
	input_active := FALSE;
END_IF

CONVERSION_this.is_active := 	(
						CONVERSION_this.status = ANALOG_ACTUATOR_STATUS_ACTIVATING
						AND
						(
							input_active
							OR
							NOT CONVERSION_this.has_di_active
						)
						AND
						(
							timer_is_expired(CONVERSION_this.timer)
							OR
							CONVERSION_this.has_di_active
						)
					)
					OR
					CONVERSION_this.status = ANALOG_ACTUATOR_STATUS_ACTIVE
					;

CONVERSION_this.is_inactive := (
						CONVERSION_this.status = ANALOG_ACTUATOR_STATUS_DEACTIVATING
						AND
						NOT input_active
						AND
						(
							timer_is_expired(CONVERSION_this.timer)
							OR
							CONVERSION_this.has_di_active
						)
					)
					OR
					CONVERSION_this.status = ANALOG_ACTUATOR_STATUS_INACTIVE
					;

END_FUNCTION

// ---- POUs/AFL extensions/analog_actuator/private/analog_actuator_submit_command.TcPOU
(* Function that executes the command assigned to the analog_actuator
	specified by the parameter 'this' *)
FUNCTION analog_actuator_submit_command : VOID


VAR
	inital_physical_value: 	LREAL;
END_VAR
(*All VAR_IN_OUT variables have been moved to the end of the declaration due to compatibility reasons*)
VAR_IN_OUT
    CONVERSION_this:	analog_actuator;	(* Instance to which the method applies *)
END_VAR

CASE CONVERSION_this.command OF
    ANALOG_ACTUATOR_CMD_ACTIVATE:
        CASE CONVERSION_this.status OF
			ANALOG_ACTUATOR_STATUS_INIT,
			ANALOG_ACTUATOR_STATUS_DEACTIVATING,
            ANALOG_ACTUATOR_STATUS_INACTIVE:
				inital_physical_value := CONVERSION_this.ao_setpoint^.physical_value;
				analog_output_physical_write(physical_value := CONVERSION_this.analog_physical_command, CONVERSION_this := CONVERSION_this.ao_setpoint^);	(*todo: to consider also percent write*)
				IF CONVERSION_this.has_do_activate
				THEN
					digital_output_set(CONVERSION_this.do_activate^);
				END_IF
                CONVERSION_this.status := ANALOG_ACTUATOR_STATUS_ACTIVATING;
                timer_restart(CONVERSION_this.active_time, CONVERSION_this.timer);

			ANALOG_ACTUATOR_STATUS_ACTIVE:	(*todo: what to do when change analog output setpoint after activate? *)

				inital_physical_value := CONVERSION_this.ao_setpoint^.physical_value;
				analog_output_physical_write(physical_value := CONVERSION_this.analog_physical_command, CONVERSION_this := CONVERSION_this.ao_setpoint^);	(*todo: to consider also percent write*)
				IF CONVERSION_this.has_do_activate
				THEN
					digital_output_set(CONVERSION_this.do_activate^);
				END_IF

				IF 	CONVERSION_this.analog_physical_command
					=
					inital_physical_value
				THEN
					CONVERSION_this.operational_command := ANALOG_ACTUATOR_CMD_NONE;
					CONVERSION_this.test.command := ANALOG_ACTUATOR_TEST_CMD_IDLE;
					CONVERSION_this.command := ANALOG_ACTUATOR_CMD_NONE;
				ELSE
	                CONVERSION_this.status := ANALOG_ACTUATOR_STATUS_ACTIVATING;
	                timer_restart(CONVERSION_this.active_time, CONVERSION_this.timer);
				END_IF
			ELSE
				CONVERSION_this.command := ANALOG_ACTUATOR_CMD_NONE;

        END_CASE;

    ANALOG_ACTUATOR_CMD_DEACTIVATE:
        CASE CONVERSION_this.status OF
			ANALOG_ACTUATOR_STATUS_INIT,
			ANALOG_ACTUATOR_STATUS_ACTIVATING,
            ANALOG_ACTUATOR_STATUS_ACTIVE:
				inital_physical_value := CONVERSION_this.ao_setpoint^.physical_value;
				analog_output_physical_write(physical_value := 0, CONVERSION_this := CONVERSION_this.ao_setpoint^);	(*todo: to consider also percent write*)

				IF CONVERSION_this.has_do_activate
				THEN
					digital_output_reset(CONVERSION_this.do_activate^);
				END_IF
                CONVERSION_this.status := ANALOG_ACTUATOR_STATUS_DEACTIVATING;
                timer_restart(CONVERSION_this.inactive_time, CONVERSION_this.timer);

			ANALOG_ACTUATOR_STATUS_INACTIVE:
				analog_output_physical_write(physical_value := 0, CONVERSION_this := CONVERSION_this.ao_setpoint^);	(*todo: to consider also percent write*)
				IF CONVERSION_this.has_do_activate
				THEN
					digital_output_reset(CONVERSION_this.do_activate^);
				END_IF

				CONVERSION_this.operational_command := ANALOG_ACTUATOR_CMD_NONE;
				CONVERSION_this.test.command := ANALOG_ACTUATOR_TEST_CMD_IDLE;
				CONVERSION_this.command := ANALOG_ACTUATOR_CMD_NONE;

			ELSE
				CONVERSION_this.command := ANALOG_ACTUATOR_CMD_NONE;

        END_CASE;

END_CASE;

IF	CONVERSION_this.command = ANALOG_ACTUATOR_CMD_NONE
THEN

	IF	descriptor_get_mode(CONVERSION_this.descriptor) = MODE_OPERATIONAL
	THEN
		CONVERSION_this.operational_command := ANALOG_ACTUATOR_CMD_NONE;
	END_IF

	CONVERSION_this.test.command := ANALOG_ACTUATOR_TEST_CMD_IDLE;

END_IF

END_FUNCTION

// ---- POUs/AFL extensions/analog_actuator/private/analog_actuator_set_snapshot.TcPOU
(* Dipslays a analog_actuator message *)
FUNCTION analog_actuator_set_snapshot : VOID
VAR_INPUT
    errorID_1:	DINT;			(* Field for specify the fault codes or enter
								   more message info *)
    errorID_2:	DINT;			(* Field for specify the fault codes or enter
								   more message info *)
    errorID_3:	DINT;			(* Field for specify the fault codes or enter
								   more message info *)
END_VAR

VAR
	owner:			POINTER TO analog_actuator;
END_VAR
(*All VAR_IN_OUT variables have been moved to the end of the declaration due to compatibility reasons*)
VAR_IN_OUT
    CONVERSION_this:			analog_actuator_snapshot;
								(* analog_actuator snapshot reference *)
END_VAR

owner := CONVERSION_this.message.CONVERSION_private.owner;

IF message_set(errorID_1, errorID_2, errorID_3, CONVERSION_this.message)
THEN
    CONVERSION_this.status := owner^.status;
    CONVERSION_this.command := owner^.command;
    CONVERSION_this.is_active := owner^.is_active;
    CONVERSION_this.is_inactive := owner^.is_inactive;
END_IF

END_FUNCTION

// ---- POUs/AFL extensions/analog_actuator/commands/analog_actuator_activate_physical_value.TcPOU
(*$
	Sends an activation command to the instance <b><i>this</i></b>, i.e.
	requests the instance to activate the linked <a href="#digital_output_object"><i>digital_output</i></a> <br/>	
	to reach the status <a href="#analog_actuator_status_enum"><i>ANALOG_ACTUATOR_STATUS_ACTIVE</i></a>.
	The command is accepted only in <a href="#mode_enum"><i>MODE_OPERATIONAL</i></a>, the object is not faulted
	and the fault reaction is <a href="#analog_actuator_fault_reaction_enum"><i>ANALOG_ACTUATOR_FAULT_REACTION_IGNORE</i></a>.<br/>
	The method returns <i>TRUE</i> if the command is accepted, otherwise it returns <i>FALSE</i>.
$*)
FUNCTION analog_actuator_activate_physical_value : BOOL
VAR_INPUT
	physical_value:		REAL;			(*$ Physical writing value $*)
END_VAR
VAR_IN_OUT
    CONVERSION_this:		analog_actuator;	(*$ Instance to which the method applies $*)
END_VAR

IF	NOT (descriptor_mode_is_operational(CONVERSION_this.descriptor)
		OR
		descriptor_mode_is_test(CONVERSION_this.descriptor))
	OR	(
			(	descriptor_is_not_ready(CONVERSION_this.descriptor)
				AND
				CONVERSION_this.fault_reaction <> ANALOG_ACTUATOR_FAULT_REACTION_IGNORE	)
		)
THEN
	analog_actuator_activate_physical_value := FALSE;					(* command rejected *)
  	RETURN;
END_IF

CONVERSION_this.operational_command := ANALOG_ACTUATOR_CMD_ACTIVATE;
CONVERSION_this.analog_physical_command := physical_value;
analog_actuator_activate_physical_value := TRUE;						(* command accepted *)

END_FUNCTION

